LIN {X 0,Y 418.536,Z 472.34,A -85,B 0,C 180,E1 -10078.075,E2 -10078.075} C_VEL
LIN {X 0,Y 418.665,Z 472.33,A -85,B 0,C 180,E1 -10080,E2 -10080} C_VEL
LIN {X 0,Y 418.503,Z 472.347,A -85,B 0,C 180,E1 -10082.888,E2 -10082.888} C_VEL
LIN {X 0,Y 418.524,Z 472.35,A -85,B 0,C 180,E1 -10085.783,E2 -10085.783} C_VEL
LIN {X 0,Y 418.391,Z 472.364,A -85,B 0,C 180,E1 -10088.695,E2 -10088.695} C_VEL
LIN {X 0,Y 418.307,Z 472.371,A -85,B 0,C 180,E1 -10091.631,E2 -10091.631} C_VEL
LIN {X 0,Y 418.293,Z 472.377,A -85,B 0,C 180,E1 -10094.597,E2 -10094.597} C_VEL
LIN {X 0,Y 418.279,Z 472.366,A -85,B 0,C 180,E1 -10097.604,E2 -10097.604} C_VEL
LIN {X 0,Y 418.242,Z 472.376,A -85,B 0,C 180,E1 -10100.663,E2 -10100.663} C_VEL
LIN {X 0,Y 418.28,Z 472.382,A -85,B 0,C 180,E1 -10103.782,E2 -10103.782} C_VEL
LIN {X 0,Y 418.303,Z 472.362,A -85,B 0,C 180,E1 -10107.071,E2 -10107.071} C_VEL
LIN {X 0,Y 418.256,Z 472.383,A -85,B 0,C 180,E1 -10110.271,E2 -10110.271} C_VEL
LIN {X 0,Y 418.243,Z 472.378,A -85,B 0,C 180,E1 -10113.678,E2 -10113.678} C_VEL
LIN {X 0,Y 418.24,Z 472.385,A -85,B 0,C 180,E1 -10117.224,E2 -10117.224} C_VEL
LIN {X 0,Y 418.25,Z 472.386,A -85,B 0,C 180,E1 -10119.682,E2 -10119.682} C_VEL
LIN {X 0,Y 418.225,Z 472.377,A -85,B 0,C 180,E1 -10122.322,E2 -10122.322} C_VEL
LIN {X 0,Y 418.254,Z 472.371,A -85,B 0,C 180,E1 -10125.113,E2 -10125.113} C_VEL
LIN {X 0,Y 418.289,Z 472.38,A -85,B 0,C 180,E1 -10127.774,E2 -10127.774} C_VEL
LIN {X 0,Y 418.262,Z 472.385,A -85,B 0,C 180,E1 -10131.56,E2 -10131.56} C_VEL
LIN {X 0,Y 418.258,Z 472.386,A -85,B 0,C 180,E1 -10135.16,E2 -10135.16} C_VEL
LIN {X 0,Y 418.282,Z 472.582,A -85,B 0,C 180,E1 -10137.69,E2 -10137.69} C_VEL
LIN {X 0,Y 421.773,Z 487.467,A -85,B 0,C 180,E1 -10140.305,E2 -10140.305} C_VEL
LIN {X 0,Y 423.139,Z 494.876,A -85,B 0,C 180,E1 -10141.54,E2 -10141.54} C_VEL
LIN {X 0,Y 421.976,Z 513.448,A -85,B 0,C 180,E1 -10144.341,E2 -10144.341} C_VEL
LIN {X 0,Y 420.64,Z 535.68,A -85,B 0,C 180,E1 -10147.66,E2 -10147.66} C_VEL
LIN {X 0,Y 419.505,Z 557.237,A -85,B 0,C 180,E1 -10150.87,E2 -10150.87} C_VEL
LIN {X 0,Y 422.696,Z 586.903,A -85,B 0,C 180,E1 -10151.56,E2 -10151.56} C_VEL
LIN {X 0,Y 423.368,Z 594.694,A -85,B 0,C 180,E1 -10151.724,E2 -10151.724} C_VEL
LIN {X 0,Y 422.593,Z 667.918,A -85,B 0,C 180,E1 -10152.987,E2 -10152.987} C_VEL
LIN {X 0,Y 422.008,Z 681.219,A -85,B 0,C 180,E1 -10153.399,E2 -10153.399} C_VEL
LIN {X 0,Y 421.231,Z 694.57,A -85,B 0,C 180,E1 -10154.021,E2 -10154.021} C_VEL
LIN {X 0,Y 420.554,Z 705.824,A -85,B 0,C 180,E1 -10154.74,E2 -10154.74} C_VEL
LIN {X 0,Y 419.697,Z 717.543,A -85,B 0,C 180,E1 -10155.701,E2 -10155.701} C_VEL
LIN {X 0,Y 419.002,Z 727.885,A -85,B 0,C 180,E1 -10156.761,E2 -10156.761} C_VEL
LIN {X 0,Y 418.593,Z 735.017,A -85,B 0,C 180,E1 -10157.64,E2 -10157.64} C_VEL
LIN {X 0,Y 418.002,Z 744.878,A -85,B 0,C 180,E1 -10159.097,E2 -10159.097} C_VEL
LIN {X 0,Y 417.68,Z 752.774,A -85,B 0,C 180,E1 -10160.558,E2 -10160.558} C_VEL
LIN {X 0,Y 417.506,Z 760.077,A -85,B 0,C 180,E1 -10162.261,E2 -10162.261} C_VEL
LIN {X 0,Y 417.494,Z 764.689,A -85,B 0,C 180,E1 -10163.63,E2 -10163.63} C_VEL
LIN {X 0,Y 417.619,Z 768.711,A -85,B 0,C 180,E1 -10165.173,E2 -10165.173} C_VEL
LIN {X 0,Y 417.674,Z 770.646,A -85,B 0,C 180,E1 -10166.141,E2 -10166.141} C_VEL
LIN {X 0,Y 417.648,Z 772.089,A -85,B 0,C 180,E1 -10167.106,E2 -10167.106} C_VEL
LIN {X 0,Y 417.907,Z 773.786,A -85,B 0,C 180,E1 -10169.036,E2 -10169.036} C_VEL
LIN {X 0,Y 417.924,Z 774.012,A -85,B 0,C 180,E1 -10170,E2 -10170} C_VEL
LIN {X 0,Y 417.907,Z 773.785,A -85,B 0,C 180,E1 -10170.964,E2 -10170.964} C_VEL
LIN {X 0,Y 417.648,Z 772.089,A -85,B 0,C 180,E1 -10172.894,E2 -10172.894} C_VEL
LIN {X 0,Y 417.674,Z 770.645,A -85,B 0,C 180,E1 -10173.859,E2 -10173.859} C_VEL
LIN {X 0,Y 417.534,Z 767.586,A -85,B 0,C 180,E1 -10175.312,E2 -10175.312} C_VEL
LIN {X 0,Y 417.475,Z 763.466,A -85,B 0,C 180,E1 -10176.767,E2 -10176.767} C_VEL
LIN {X 0,Y 417.531,Z 757.153,A -85,B 0,C 180,E1 -10178.469,E2 -10178.469} C_VEL
LIN {X 0,Y 417.723,Z 750.287,A -85,B 0,C 180,E1 -10179.93,E2 -10179.93} C_VEL
LIN {X 0,Y 418.17,Z 741.814,A -85,B 0,C 180,E1 -10181.389,E2 -10181.389} C_VEL
LIN {X 0,Y 418.764,Z 733.161,A -85,B 0,C 180,E1 -10182.602,E2 -10182.602} C_VEL
LIN {X 0,Y 419.355,Z 722.483,A -85,B 0,C 180,E1 -10183.816,E2 -10183.816} C_VEL
LIN {X 0,Y 420.141,Z 710.52,A -85,B 0,C 180,E1 -10184.903,E2 -10184.903} C_VEL
LIN {X 0,Y 421.03,Z 698.539,A -85,B 0,C 180,E1 -10185.738,E2 -10185.738} C_VEL
LIN {X 0,Y 421.752,Z 686.096,A -85,B 0,C 180,E1 -10186.394,E2 -10186.394} C_VEL
LIN {X 0,Y 422.39,Z 673.352,A -85,B 0,C 180,E1 -10186.866,E2 -10186.866} C_VEL
LIN {X 0,Y 422.723,Z 658.22,A -85,B 0,C 180,E1 -10187.194,E2 -10187.194} C_VEL
LIN {X 0,Y 423.312,Z 592.38,A -85,B 0,C 180,E1 -10188.314,E2 -10188.314} C_VEL
LIN {X 0,Y 419.505,Z 557.278,A -85,B 0,C 180,E1 -10189.121,E2 -10189.121} C_VEL
LIN {X 0,Y 420.722,Z 533.922,A -85,B 0,C 180,E1 -10192.594,E2 -10192.594} C_VEL
LIN {X 0,Y 422.251,Z 509.398,A -85,B 0,C 180,E1 -10196.258,E2 -10196.258} C_VEL
LIN {X 0,Y 423.139,Z 494.649,A -85,B 0,C 180,E1 -10198.486,E2 -10198.486} C_VEL
LIN {X 0,Y 421.349,Z 485.456,A -85,B 0,C 180,E1 -10200.025,E2 -10200.025} C_VEL
LIN {X 0,Y 418.28,Z 472.498,A -85,B 0,C 180,E1 -10202.346,E2 -10202.346} C_VEL
LIN {X 0,Y 418.257,Z 472.387,A -85,B 0,C 180,E1 -10204.84,E2 -10204.84} C_VEL
LIN {X 0,Y 418.262,Z 472.385,A -85,B 0,C 180,E1 -10208.44,E2 -10208.44} C_VEL
LIN {X 0,Y 418.289,Z 472.381,A -85,B 0,C 180,E1 -10212.226,E2 -10212.226} C_VEL
LIN {X 0,Y 418.247,Z 472.37,A -85,B 0,C 180,E1 -10215.11,E2 -10215.11} C_VEL
LIN {X 0,Y 418.235,Z 472.376,A -85,B 0,C 180,E1 -10217.766,E2 -10217.766} C_VEL
LIN {X 0,Y 418.254,Z 472.381,A -85,B 0,C 180,E1 -10220.617,E2 -10220.617} C_VEL
LIN {X 0,Y 418.24,Z 472.387,A -85,B 0,C 180,E1 -10223.975,E2 -10223.975} C_VEL
LIN {X 0,Y 418.251,Z 472.375,A -85,B 0,C 180,E1 -10227.155,E2 -10227.155} C_VEL
LIN {X 0,Y 418.268,Z 472.379,A -85,B 0,C 180,E1 -10230.838,E2 -10230.838} C_VEL
LIN {X 0,Y 418.264,Z 472.371,A -85,B 0,C 180,E1 -10234.095,E2 -10234.095} C_VEL
LIN {X 0,Y 418.23,Z 472.385,A -85,B 0,C 180,E1 -10237.263,E2 -10237.263} C_VEL
LIN {X 0,Y 418.275,Z 472.364,A -85,B 0,C 180,E1 -10240.364,E2 -10240.364} C_VEL
LIN {X 0,Y 418.308,Z 472.37,A -85,B 0,C 180,E1 -10243.404,E2 -10243.404} C_VEL
LIN {X 0,Y 418.337,Z 472.37,A -85,B 0,C 180,E1 -10246.999,E2 -10246.999} C_VEL
LIN {X 0,Y 418.333,Z 472.369,A -85,B 0,C 180,E1 -10250.328,E2 -10250.328} C_VEL
LIN {X 0,Y 418.486,Z 472.352,A -85,B 0,C 180,E1 -10253.249,E2 -10253.249} C_VEL
LIN {X 0,Y 418.337,Z 472.361,A -85,B 0,C 180,E1 -10255.182,E2 -10255.182} C_VEL
LIN {X 0,Y 418.536,Z 472.346,A -85,B 0,C 180,E1 -10258.075,E2 -10258.075} C_VEL
LIN {X 0,Y 418.665,Z 472.332,A -85,B 0,C 180,E1 -10260,E2 -10260} C_VEL
LIN {X 0,Y 418.503,Z 472.345,A -85,B 0,C 180,E1 -10262.888,E2 -10262.888} C_VEL
LIN {X 0,Y 418.484,Z 472.355,A -85,B 0,C 180,E1 -10266.615,E2 -10266.615} C_VEL
LIN {X 0,Y 418.333,Z 472.361,A -85,B 0,C 180,E1 -10269.672,E2 -10269.672} C_VEL
LIN {X 0,Y 418.338,Z 472.374,A -85,B 0,C 180,E1 -10273.001,E2 -10273.001} C_VEL
LIN {X 0,Y 418.304,Z 472.371,A -85,B 0,C 180,E1 -10276.736,E2 -10276.736} C_VEL
LIN {X 0,Y 418.263,Z 472.381,A -85,B 0,C 180,E1 -10279.791,E2 -10279.791} C_VEL
LIN {X 0,Y 418.23,Z 472.381,A -85,B 0,C 180,E1 -10282.737,E2 -10282.737} C_VEL
LIN {X 0,Y 418.264,Z 472.381,A -85,B 0,C 180,E1 -10285.905,E2 -10285.905} C_VEL
LIN {X 0,Y 418.268,Z 472.36,A -85,B 0,C 180,E1 -10289.162,E2 -10289.162} C_VEL
LIN {X 0,Y 418.252,Z 472.37,A -85,B 0,C 180,E1 -10292.845,E2 -10292.845} C_VEL
LIN {X 0,Y 418.243,Z 472.385,A -85,B 0,C 180,E1 -10296.239,E2 -10296.239} C_VEL
LIN {X 0,Y 418.24,Z 472.361,A -85,B 0,C 180,E1 -10299.683,E2 -10299.683} C_VEL
LIN {X 0,Y 418.225,Z 472.38,A -85,B 0,C 180,E1 -10302.322,E2 -10302.322} C_VEL
LIN {X 0,Y 418.235,Z 472.385,A -85,B 0,C 180,E1 -10305.11,E2 -10305.11} C_VEL
LIN {X 0,Y 418.239,Z 472.372,A -85,B 0,C 180,E1 -10307.768,E2 -10307.768} C_VEL
LIN {X 0,Y 418.259,Z 472.385,A -85,B 0,C 180,E1 -10310.619,E2 -10310.619} C_VEL
LIN {X 0,Y 418.244,Z 472.359,A -85,B 0,C 180,E1 -10313.977,E2 -10313.977} C_VEL
LIN {X 0,Y 418.257,Z 472.359,A -85,B 0,C 180,E1 -10317.157,E2 -10317.157} C_VEL
LIN {X 0,Y 418.268,Z 472.378,A -85,B 0,C 180,E1 -10320.896,E2 -10320.896} C_VEL
LIN {X 0,Y 418.271,Z 472.368,A -85,B 0,C 180,E1 -10324.097,E2 -10324.097} C_VEL
LIN {X 0,Y 418.239,Z 472.371,A -85,B 0,C 180,E1 -10327.265,E2 -10327.265} C_VEL
LIN {X 0,Y 418.324,Z 472.346,A -85,B 0,C 180,E1 -10330.877,E2 -10330.877} C_VEL
LIN {X 0,Y 418.375,Z 472.623,A -85,B 0,C 180,E1 -10331.261,E2 -10331.261} C_VEL
LIN {X 0,Y 418.655,Z 473.76,A -85,B 0,C 180,E1 -10331.401,E2 -10331.401} C_VEL
LIN {X 0,Y 424.299,Z 488.537,A -85,B 0,C 180,E1 -10331.94,E2 -10331.94} C_VEL
LIN {X 0,Y 423.71,Z 551.851,A -85,B 0,C 180,E1 -10333.033,E2 -10333.033} C_VEL
LIN {X 0,Y 423.641,Z 564.47,A -85,B 0,C 180,E1 -10333.403,E2 -10333.403} C_VEL
LIN {X 0,Y 423.281,Z 577.262,A -85,B 0,C 180,E1 -10333.977,E2 -10333.977} C_VEL
LIN {X 0,Y 422.895,Z 589.004,A -85,B 0,C 180,E1 -10334.702,E2 -10334.702} C_VEL
LIN {X 0,Y 422.287,Z 599.691,A -85,B 0,C 180,E1 -10335.544,E2 -10335.544} C_VEL
LIN {X 0,Y 421.612,Z 610.545,A -85,B 0,C 180,E1 -10336.627,E2 -10336.627} C_VEL
LIN {X 0,Y 420.921,Z 621.071,A -85,B 0,C 180,E1 -10337.954,E2 -10337.954} C_VEL
LIN {X 0,Y 420.413,Z 628.814,A -85,B 0,C 180,E1 -10339.16,E2 -10339.16} C_VEL
LIN {X 0,Y 419.767,Z 636.5,A -85,B 0,C 180,E1 -10340.63,E2 -10340.63} C_VEL
LIN {X 0,Y 419.323,Z 642.255,A -85,B 0,C 180,E1 -10342.003,E2 -10342.003} C_VEL
LIN {X 0,Y 419.063,Z 646.526,A -85,B 0,C 180,E1 -10343.258,E2 -10343.258} C_VEL
LIN {X 0,Y 418.621,Z 650.42,A -85,B 0,C 180,E1 -10344.702,E2 -10344.702} C_VEL
LIN {X 0,Y 418.398,Z 652.498,A -85,B 0,C 180,E1 -10345.73,E2 -10345.73} C_VEL
LIN {X 0,Y 417.639,Z 653.952,A -85,B 0,C 180,E1 -10346.509,E2 -10346.509} C_VEL
LIN {X 0,Y 414.72,Z 655.903,A -85,B 0,C 180,E1 -10347.785,E2 -10347.785} C_VEL
LIN {X 0,Y 412.318,Z 656.955,A -85,B 0,C 180,E1 -10348.826,E2 -10348.826} C_VEL
LIN {X 0,Y 411.309,Z 657.36,A -85,B 0,C 180,E1 -10349.635,E2 -10349.635} C_VEL
LIN {X 0,Y 411.236,Z 657.406,A -85,B 0,C 180,E1 -10349.91,E2 -10349.91} C_VEL
LIN {X 0,Y 411.256,Z 657.243,A -85,B 0,C 180,E1 -10350.979,E2 -10350.979} C_VEL
LIN {X 0,Y 411.181,Z 656.69,A -85,B 0,C 180,E1 -10351.959,E2 -10351.959} C_VEL
LIN {X 0,Y 411.339,Z 655.735,A -85,B 0,C 180,E1 -10352.938,E2 -10352.938} C_VEL
LIN {X 0,Y 411.318,Z 654.429,A -85,B 0,C 180,E1 -10353.919,E2 -10353.919} C_VEL
LIN {X 0,Y 411.614,Z 651.618,A -85,B 0,C 180,E1 -10355.388,E2 -10355.388} C_VEL
LIN {X 0,Y 412.065,Z 647.796,A -85,B 0,C 180,E1 -10356.857,E2 -10356.857} C_VEL
LIN {X 0,Y 412.366,Z 642.722,A -85,B 0,C 180,E1 -10358.378,E2 -10358.378} C_VEL
LIN {X 0,Y 412.913,Z 636.698,A -85,B 0,C 180,E1 -10359.8,E2 -10359.8} C_VEL
LIN {X 0,Y 413.612,Z 628.922,A -85,B 0,C 180,E1 -10361.268,E2 -10361.268} C_VEL
LIN {X 0,Y 414.28,Z 619.255,A -85,B 0,C 180,E1 -10362.74,E2 -10362.74} C_VEL
LIN {X 0,Y 414.951,Z 610.219,A -85,B 0,C 180,E1 -10363.841,E2 -10363.841} C_VEL
LIN {X 0,Y 415.667,Z 599.725,A -85,B 0,C 180,E1 -10364.873,E2 -10364.873} C_VEL
LIN {X 0,Y 416.209,Z 588.069,A -85,B 0,C 180,E1 -10365.787,E2 -10365.787} C_VEL
LIN {X 0,Y 416.646,Z 576.642,A -85,B 0,C 180,E1 -10366.474,E2 -10366.474} C_VEL
LIN {X 0,Y 416.932,Z 563.782,A -85,B 0,C 180,E1 -10367.03,E2 -10367.03} C_VEL
LIN {X 0,Y 416.972,Z 551.522,A -85,B 0,C 180,E1 -10367.376,E2 -10367.376} C_VEL
LIN {X 0,Y 417.43,Z 489.383,A -85,B 0,C 180,E1 -10368.47,E2 -10368.47} C_VEL
LIN {X 0,Y 411.516,Z 474.325,A -85,B 0,C 180,E1 -10369.052,E2 -10369.052} C_VEL
LIN {X 0,Y 411.297,Z 473.373,A -85,B 0,C 180,E1 -10369.236,E2 -10369.236} C_VEL
LIN {X 0,Y 411.204,Z 473.25,A -85,B 0,C 180,E1 -10373.147,E2 -10373.147} C_VEL
LIN {X 0,Y 411.238,Z 473.237,A -85,B 0,C 180,E1 -10376.38,E2 -10376.38} C_VEL
LIN {X 0,Y 411.2,Z 473.263,A -85,B 0,C 180,E1 -10379.712,E2 -10379.712} C_VEL
LIN {X 0,Y 411.205,Z 473.259,A -85,B 0,C 180,E1 -10383.155,E2 -10383.155} C_VEL
LIN {X 0,Y 411.194,Z 473.256,A -85,B 0,C 180,E1 -10386.552,E2 -10386.552} C_VEL
LIN {X 0,Y 411.214,Z 473.262,A -85,B 0,C 180,E1 -10389.727,E2 -10389.727} C_VEL
LIN {X 0,Y 411.174,Z 473.253,A -85,B 0,C 180,E1 -10393.132,E2 -10393.132} C_VEL
LIN {X 0,Y 411.165,Z 473.267,A -85,B 0,C 180,E1 -10395.88,E2 -10395.88} C_VEL
LIN {X 0,Y 411.159,Z 473.254,A -85,B 0,C 180,E1 -10398.771,E2 -10398.771} C_VEL
LIN {X 0,Y 411.191,Z 473.256,A -85,B 0,C 180,E1 -10402.026,E2 -10402.026} C_VEL
LIN {X 0,Y 411.2,Z 473.258,A -85,B 0,C 180,E1 -10405.666,E2 -10405.666} C_VEL
LIN {X 0,Y 411.191,Z 473.233,A -85,B 0,C 180,E1 -10409.152,E2 -10409.152} C_VEL
LIN {X 0,Y 411.253,Z 473.247,A -85,B 0,C 180,E1 -10412.522,E2 -10412.522} C_VEL
LIN {X 0,Y 411.219,Z 473.257,A -85,B 0,C 180,E1 -10415.784,E2 -10415.784} C_VEL
LIN {X 0,Y 411.188,Z 473.259,A -85,B 0,C 180,E1 -10418.965,E2 -10418.965} C_VEL
LIN {X 0,Y 411.244,Z 473.252,A -85,B 0,C 180,E1 -10422.084,E2 -10422.084} C_VEL
LIN {X 0,Y 411.252,Z 473.251,A -85,B 0,C 180,E1 -10425.147,E2 -10425.147} C_VEL
LIN {X 0,Y 411.276,Z 473.25,A -85,B 0,C 180,E1 -10428.167,E2 -10428.167} C_VEL
LIN {X 0,Y 411.473,Z 473.223,A -85,B 0,C 180,E1 -10432.146,E2 -10432.146} C_VEL
LIN {X 0,Y 411.466,Z 473.226,A -85,B 0,C 180,E1 -10434.118,E2 -10434.118} C_VEL
LIN {X 0,Y 411.505,Z 473.216,A -85,B 0,C 180,E1 -10438.042,E2 -10438.042} C_VEL
LIN {X 0,Y 411.635,Z 473.206,A -85,B 0,C 180,E1 -10440,E2 -10440} C_VEL
LIN {X 0,Y 411.458,Z 473.225,A -85,B 0,C 180,E1 -10442.937,E2 -10442.937} C_VEL
LIN {X 0,Y 411.483,Z 473.226,A -85,B 0,C 180,E1 -10445.882,E2 -10445.882} C_VEL
LIN {X 0,Y 411.346,Z 473.242,A -85,B 0,C 180,E1 -10448.845,E2 -10448.845} C_VEL
LIN {X 0,Y 411.276,Z 473.249,A -85,B 0,C 180,E1 -10451.833,E2 -10451.833} C_VEL
LIN {X 0,Y 411.251,Z 473.255,A -85,B 0,C 180,E1 -10454.853,E2 -10454.853} C_VEL
LIN {X 0,Y 411.244,Z 473.238,A -85,B 0,C 180,E1 -10457.915,E2 -10457.915} C_VEL
LIN {X 0,Y 411.188,Z 473.256,A -85,B 0,C 180,E1 -10461.035,E2 -10461.035} C_VEL
LIN {X 0,Y 411.219,Z 473.257,A -85,B 0,C 180,E1 -10464.216,E2 -10464.216} C_VEL
LIN {X 0,Y 411.253,Z 473.242,A -85,B 0,C 180,E1 -10467.478,E2 -10467.478} C_VEL
LIN {X 0,Y 411.194,Z 473.262,A -85,B 0,C 180,E1 -10470.847,E2 -10470.847} C_VEL
LIN {X 0,Y 411.201,Z 473.26,A -85,B 0,C 180,E1 -10474.334,E2 -10474.334} C_VEL
LIN {X 0,Y 411.195,Z 473.258,A -85,B 0,C 180,E1 -10477.974,E2 -10477.974} C_VEL
LIN {X 0,Y 411.178,Z 473.265,A -85,B 0,C 180,E1 -10480.505,E2 -10480.505} C_VEL
LIN {X 0,Y 411.168,Z 473.25,A -85,B 0,C 180,E1 -10483.134,E2 -10483.134} C_VEL
LIN {X 0,Y 411.232,Z 473.253,A -85,B 0,C 180,E1 -10485.872,E2 -10485.872} C_VEL
LIN {X 0,Y 411.207,Z 473.254,A -85,B 0,C 180,E1 -10488.765,E2 -10488.765} C_VEL
LIN {X 0,Y 411.201,Z 473.264,A -85,B 0,C 180,E1 -10492.028,E2 -10492.028} C_VEL
LIN {X 0,Y 411.204,Z 473.261,A -85,B 0,C 180,E1 -10495.667,E2 -10495.667} C_VEL
LIN {X 0,Y 411.241,Z 473.427,A -85,B 0,C 180,E1 -10497.358,E2 -10497.358} C_VEL
LIN {X 0,Y 414.904,Z 489.081,A -85,B 0,C 180,E1 -10500.172,E2 -10500.172} C_VEL
LIN {X 0,Y 416.266,Z 496.273,A -85,B 0,C 180,E1 -10501.395,E2 -10501.395} C_VEL
LIN {X 0,Y 415.073,Z 514.231,A -85,B 0,C 180,E1 -10504.152,E2 -10504.152} C_VEL
LIN {X 0,Y 413.65,Z 536.399,A -85,B 0,C 180,E1 -10507.526,E2 -10507.526} C_VEL
LIN {X 0,Y 412.575,Z 556.343,A -85,B 0,C 180,E1 -10510.545,E2 -10510.545} C_VEL
LIN {X 0,Y 415.931,Z 587.374,A -85,B 0,C 180,E1 -10511.274,E2 -10511.274} C_VEL
LIN {X 0,Y 416.594,Z 595.875,A -85,B 0,C 180,E1 -10511.454,E2 -10511.454} C_VEL
LIN {X 0,Y 415.799,Z 666.93,A -85,B 0,C 180,E1 -10512.7,E2 -10512.7} C_VEL
LIN {X 0,Y 415.202,Z 680.228,A -85,B 0,C 180,E1 -10513.119,E2 -10513.119} C_VEL
LIN {X 0,Y 414.376,Z 693.573,A -85,B 0,C 180,E1 -10513.749,E2 -10513.749} C_VEL
LIN {X 0,Y 413.631,Z 704.819,A -85,B 0,C 180,E1 -10514.478,E2 -10514.478} C_VEL
LIN {X 0,Y 412.746,Z 716.537,A -85,B 0,C 180,E1 -10515.455,E2 -10515.455} C_VEL
LIN {X 0,Y 412.018,Z 726.405,A -85,B 0,C 180,E1 -10516.478,E2 -10516.478} C_VEL
LIN {X 0,Y 411.638,Z 734.018,A -85,B 0,C 180,E1 -10517.427,E2 -10517.427} C_VEL
LIN {X 0,Y 411.052,Z 742.351,A -85,B 0,C 180,E1 -10518.661,E2 -10518.661} C_VEL
LIN {X 0,Y 410.637,Z 750.568,A -85,B 0,C 180,E1 -10520.146,E2 -10520.146} C_VEL
LIN {X 0,Y 410.451,Z 757.194,A -85,B 0,C 180,E1 -10521.632,E2 -10521.632} C_VEL
LIN {X 0,Y 410.418,Z 763.067,A -85,B 0,C 180,E1 -10523.312,E2 -10523.312} C_VEL
LIN {X 0,Y 410.546,Z 767.714,A -85,B 0,C 180,E1 -10525.09,E2 -10525.09} C_VEL
LIN {X 0,Y 410.635,Z 769.655,A -85,B 0,C 180,E1 -10526.075,E2 -10526.075} C_VEL
LIN {X 0,Y 410.604,Z 771.098,A -85,B 0,C 180,E1 -10527.057,E2 -10527.057} C_VEL
LIN {X 0,Y 410.88,Z 772.798,A -85,B 0,C 180,E1 -10529.02,E2 -10529.02} C_VEL
LIN {X 0,Y 410.902,Z 773.025,A -85,B 0,C 180,E1 -10530,E2 -10530} C_VEL
LIN {X 0,Y 410.881,Z 772.797,A -85,B 0,C 180,E1 -10530.98,E2 -10530.98} C_VEL
LIN {X 0,Y 410.604,Z 771.097,A -85,B 0,C 180,E1 -10532.943,E2 -10532.943} C_VEL
LIN {X 0,Y 410.635,Z 769.653,A -85,B 0,C 180,E1 -10533.925,E2 -10533.925} C_VEL
LIN {X 0,Y 410.46,Z 766.587,A -85,B 0,C 180,E1 -10535.404,E2 -10535.404} C_VEL
LIN {X 0,Y 410.421,Z 762.466,A -85,B 0,C 180,E1 -10536.884,E2 -10536.884} C_VEL
LIN {X 0,Y 410.464,Z 756.147,A -85,B 0,C 180,E1 -10538.616,E2 -10538.616} C_VEL
LIN {X 0,Y 410.665,Z 749.278,A -85,B 0,C 180,E1 -10540.103,E2 -10540.103} C_VEL
LIN {X 0,Y 411.145,Z 740.804,A -85,B 0,C 180,E1 -10541.586,E2 -10541.586} C_VEL
LIN {X 0,Y 411.774,Z 732.151,A -85,B 0,C 180,E1 -10542.819,E2 -10542.819} C_VEL
LIN {X 0,Y 412.319,Z 722.665,A -85,B 0,C 180,E1 -10543.931,E2 -10543.931} C_VEL
LIN {X 0,Y 413.112,Z 710.953,A -85,B 0,C 180,E1 -10545.036,E2 -10545.036} C_VEL
LIN {X 0,Y 414.041,Z 699.479,A -85,B 0,C 180,E1 -10545.885,E2 -10545.885} C_VEL
LIN {X 0,Y 414.765,Z 687.701,A -85,B 0,C 180,E1 -10546.551,E2 -10546.551} C_VEL
LIN {X 0,Y 415.503,Z 674.18,A -85,B 0,C 180,E1 -10547.09,E2 -10547.09} C_VEL
LIN {X 0,Y 415.893,Z 660.789,A -85,B 0,C 180,E1 -10547.422,E2 -10547.422} C_VEL
LIN {X 0,Y 416.518,Z 592.858,A -85,B 0,C 180,E1 -10548.597,E2 -10548.597} C_VEL
LIN {X 0,Y 412.55,Z 556.589,A -85,B 0,C 180,E1 -10549.433,E2 -10549.433} C_VEL
LIN {X 0,Y 412.898,Z 549.484,A -85,B 0,C 180,E1 -10550.47,E2 -10550.47} C_VEL
LIN {X 0,Y 414.285,Z 526.14,A -85,B 0,C 180,E1 -10554.025,E2 -10554.025} C_VEL
LIN {X 0,Y 415.776,Z 503.859,A -85,B 0,C 180,E1 -10557.426,E2 -10557.426} C_VEL
LIN {X 0,Y 416.271,Z 496.209,A -85,B 0,C 180,E1 -10558.606,E2 -10558.606} C_VEL
LIN {X 0,Y 414.493,Z 487.187,A -85,B 0,C 180,E1 -10560.147,E2 -10560.147} C_VEL
LIN {X 0,Y 411.226,Z 473.379,A -85,B 0,C 180,E1 -10562.661,E2 -10562.661} C_VEL
LIN {X 0,Y 411.197,Z 473.26,A -85,B 0,C 180,E1 -10565.528,E2 -10565.528} C_VEL
LIN {X 0,Y 411.227,Z 473.255,A -85,B 0,C 180,E1 -10569.222,E2 -10569.222} C_VEL
LIN {X 0,Y 411.229,Z 473.262,A -85,B 0,C 180,E1 -10572.703,E2 -10572.703} C_VEL
LIN {X 0,Y 411.167,Z 473.244,A -85,B 0,C 180,E1 -10575.88,E2 -10575.88} C_VEL
LIN {X 0,Y 411.16,Z 473.269,A -85,B 0,C 180,E1 -10578.771,E2 -10578.771} C_VEL
LIN {X 0,Y 411.206,Z 473.255,A -85,B 0,C 180,E1 -10581.83,E2 -10581.83} C_VEL
LIN {X 0,Y 411.205,Z 473.258,A -85,B 0,C 180,E1 -10585.121,E2 -10585.121} C_VEL
LIN {X 0,Y 411.162,Z 473.261,A -85,B 0,C 180,E1 -10588.002,E2 -10588.002} C_VEL
LIN {X 0,Y 411.217,Z 473.255,A -85,B 0,C 180,E1 -10591.41,E2 -10591.41} C_VEL
LIN {X 0,Y 411.231,Z 473.243,A -85,B 0,C 180,E1 -10593.619,E2 -10593.619} C_VEL
LIN {X 0,Y 411.195,Z 473.263,A -85,B 0,C 180,E1 -10596.852,E2 -10596.852} C_VEL
LIN {X 0,Y 411.207,Z 473.248,A -85,B 0,C 180,E1 -10600.05,E2 -10600.05} C_VEL
LIN {X 0,Y 411.255,Z 473.25,A -85,B 0,C 180,E1 -10603.131,E2 -10603.131} C_VEL
LIN {X 0,Y 411.297,Z 473.248,A -85,B 0,C 180,E1 -10606.896,E2 -10606.896} C_VEL
LIN {X 0,Y 411.285,Z 473.245,A -85,B 0,C 180,E1 -10610.161,E2 -10610.161} C_VEL
LIN {X 0,Y 411.449,Z 473.229,A -85,B 0,C 180,E1 -10613.133,E2 -10613.133} C_VEL
LIN {X 0,Y 411.308,Z 473.237,A -85,B 0,C 180,E1 -10615.099,E2 -10615.099} C_VEL
LIN {X 0,Y 411.505,Z 473.222,A -85,B 0,C 180,E1 -10618.043,E2 -10618.043} C_VEL
LIN {X 0,Y 411.635,Z 473.208,A -85,B 0,C 180,E1 -10620,E2 -10620} C_VEL
LIN {X 0,Y 411.459,Z 473.222,A -85,B 0,C 180,E1 -10622.937,E2 -10622.937} C_VEL
LIN {X 0,Y 411.447,Z 473.229,A -85,B 0,C 180,E1 -10626.614,E2 -10626.614} C_VEL
LIN {X 0,Y 411.285,Z 473.239,A -85,B 0,C 180,E1 -10629.839,E2 -10629.839} C_VEL
LIN {X 0,Y 411.297,Z 473.25,A -85,B 0,C 180,E1 -10633.104,E2 -10633.104} C_VEL
LIN {X 0,Y 411.249,Z 473.251,A -85,B 0,C 180,E1 -10636.889,E2 -10636.889} C_VEL
LIN {X 0,Y 411.223,Z 473.258,A -85,B 0,C 180,E1 -10639.987,E2 -10639.987} C_VEL
LIN {X 0,Y 411.196,Z 473.261,A -85,B 0,C 180,E1 -10643.148,E2 -10643.148} C_VEL
LIN {X 0,Y 411.231,Z 473.259,A -85,B 0,C 180,E1 -10646.382,E2 -10646.382} C_VEL
LIN {X 0,Y 411.204,Z 473.236,A -85,B 0,C 180,E1 -10649.713,E2 -10649.713} C_VEL
LIN {X 0,Y 411.201,Z 473.253,A -85,B 0,C 180,E1 -10653.157,E2 -10653.157} C_VEL
LIN {X 0,Y 411.19,Z 473.266,A -85,B 0,C 180,E1 -10656.554,E2 -10656.554} C_VEL
LIN {X 0,Y 411.204,Z 473.236,A -85,B 0,C 180,E1 -10659.728,E2 -10659.728} C_VEL
LIN {X 0,Y 411.169,Z 473.269,A -85,B 0,C 180,E1 -10663.134,E2 -10663.134} C_VEL
LIN {X 0,Y 411.169,Z 473.259,A -85,B 0,C 180,E1 -10665.881,E2 -10665.881} C_VEL
LIN {X 0,Y 411.163,Z 473.259,A -85,B 0,C 180,E1 -10668.772,E2 -10668.772} C_VEL
LIN {X 0,Y 411.21,Z 473.256,A -85,B 0,C 180,E1 -10671.831,E2 -10671.831} C_VEL
LIN {X 0,Y 411.21,Z 473.217,A -85,B 0,C 180,E1 -10675.122,E2 -10675.122} C_VEL
LIN {X 0,Y 411.165,Z 473.261,A -85,B 0,C 180,E1 -10678.004,E2 -10678.004} C_VEL
LIN {X 0,Y 411.218,Z 473.248,A -85,B 0,C 180,E1 -10681.411,E2 -10681.411} C_VEL
LIN {X 0,Y 411.238,Z 473.236,A -85,B 0,C 180,E1 -10683.62,E2 -10683.62} C_VEL
LIN {X 0,Y 411.204,Z 473.251,A -85,B 0,C 180,E1 -10686.853,E2 -10686.853} C_VEL
LIN {X 0,Y 411.308,Z 473.339,A -85,B 0,C 180,E1 -10690.862,E2 -10690.862} C_VEL
LIN {X 0,Y 411.456,Z 474.138,A -85,B 0,C 180,E1 -10691.031,E2 -10691.031} C_VEL
LIN {X 0,Y 417.419,Z 489.367,A -85,B 0,C 180,E1 -10691.628,E2 -10691.628} C_VEL
LIN {X 0,Y 416.975,Z 554.337,A -85,B 0,C 180,E1 -10692.782,E2 -10692.782} C_VEL
LIN {X 0,Y 416.801,Z 567.775,A -85,B 0,C 180,E1 -10693.217,E2 -10693.217} C_VEL
LIN {X 0,Y 416.499,Z 580.488,A -85,B 0,C 180,E1 -10693.835,E2 -10693.835} C_VEL
LIN {X 0,Y 416.078,Z 591.709,A -85,B 0,C 180,E1 -10694.57,E2 -10694.57} C_VEL
LIN {X 0,Y 415.34,Z 603.297,A -85,B 0,C 180,E1 -10695.547,E2 -10695.547} C_VEL
LIN {X 0,Y 414.661,Z 613.632,A -85,B 0,C 180,E1 -10696.649,E2 -10696.649} C_VEL
LIN {X 0,Y 414.05,Z 622.063,A -85,B 0,C 180,E1 -10697.751,E2 -10697.751} C_VEL
LIN {X 0,Y 413.513,Z 629.805,A -85,B 0,C 180,E1 -10698.977,E2 -10698.977} C_VEL
LIN {X 0,Y 412.835,Z 637.49,A -85,B 0,C 180,E1 -10700.471,E2 -10700.471} C_VEL
LIN {X 0,Y 412.365,Z 643.245,A -85,B 0,C 180,E1 -10701.867,E2 -10701.867} C_VEL
LIN {X 0,Y 412.086,Z 647.516,A -85,B 0,C 180,E1 -10703.144,E2 -10703.144} C_VEL
LIN {X 0,Y 411.622,Z 651.409,A -85,B 0,C 180,E1 -10704.612,E2 -10704.612} C_VEL
LIN {X 0,Y 411.327,Z 654.277,A -85,B 0,C 180,E1 -10706.081,E2 -10706.081} C_VEL
LIN {X 0,Y 411.341,Z 655.63,A -85,B 0,C 180,E1 -10707.062,E2 -10707.062} C_VEL
LIN {X 0,Y 411.181,Z 656.615,A -85,B 0,C 180,E1 -10708.041,E2 -10708.041} C_VEL
LIN {X 0,Y 411.236,Z 657.406,A -85,B 0,C 180,E1 -10709.91,E2 -10709.91} C_VEL
LIN {X 0,Y 410.586,Z 657.53,A -85,B 0,C 180,E1 -10710.729,E2 -10710.729} C_VEL
LIN {X 0,Y 407.725,Z 657.299,A -85,B 0,C 180,E1 -10712.061,E2 -10712.061} C_VEL
LIN {X 0,Y 404.908,Z 656.219,A -85,B 0,C 180,E1 -10713.398,E2 -10713.398} C_VEL
LIN {X 0,Y 404.336,Z 655.01,A -85,B 0,C 180,E1 -10714.216,E2 -10714.216} C_VEL
LIN {X 0,Y 404.666,Z 651.444,A -85,B 0,C 180,E1 -10715.981,E2 -10715.981} C_VEL
LIN {X 0,Y 405.204,Z 647.259,A -85,B 0,C 180,E1 -10717.474,E2 -10717.474} C_VEL
LIN {X 0,Y 405.646,Z 640.968,A -85,B 0,C 180,E1 -10719.222,E2 -10719.222} C_VEL
LIN {X 0,Y 406.366,Z 634.005,A -85,B 0,C 180,E1 -10720.714,E2 -10720.714} C_VEL
LIN {X 0,Y 407.065,Z 625.341,A -85,B 0,C 180,E1 -10722.21,E2 -10722.21} C_VEL
LIN {X 0,Y 407.71,Z 616.437,A -85,B 0,C 180,E1 -10723.456,E2 -10723.456} C_VEL
LIN {X 0,Y 408.441,Z 606.54,A -85,B 0,C 180,E1 -10724.575,E2 -10724.575} C_VEL
LIN {X 0,Y 409.185,Z 595.39,A -85,B 0,C 180,E1 -10725.577,E2 -10725.577} C_VEL
LIN {X 0,Y 409.639,Z 585.851,A -85,B 0,C 180,E1 -10726.266,E2 -10726.266} C_VEL
LIN {X 0,Y 409.992,Z 573.81,A -85,B 0,C 180,E1 -10726.942,E2 -10726.942} C_VEL
LIN {X 0,Y 410.182,Z 561.114,A -85,B 0,C 180,E1 -10727.448,E2 -10727.448} C_VEL
LIN {X 0,Y 410.191,Z 547.599,A -85,B 0,C 180,E1 -10727.769,E2 -10727.769} C_VEL
LIN {X 0,Y 410.737,Z 490.961,A -85,B 0,C 180,E1 -10728.771,E2 -10728.771} C_VEL
LIN {X 0,Y 404.404,Z 475.006,A -85,B 0,C 180,E1 -10729.42,E2 -10729.42} C_VEL
LIN {X 0,Y 404.228,Z 474.204,A -85,B 0,C 180,E1 -10729.625,E2 -10729.625} C_VEL
LIN {X 0,Y 404.17,Z 474.132,A -85,B 0,C 180,E1 -10733.574,E2 -10733.574} C_VEL
LIN {X 0,Y 404.184,Z 474.125,A -85,B 0,C 180,E1 -10735.766,E2 -10735.766} C_VEL
LIN {X 0,Y 404.195,Z 474.113,A -85,B 0,C 180,E1 -10737.999,E2 -10737.999} C_VEL
LIN {X 0,Y 404.139,Z 474.138,A -85,B 0,C 180,E1 -10741.557,E2 -10741.557} C_VEL
LIN {X 0,Y 404.184,Z 474.139,A -85,B 0,C 180,E1 -10745.015,E2 -10745.015} C_VEL
LIN {X 0,Y 404.156,Z 474.139,A -85,B 0,C 180,E1 -10748.756,E2 -10748.756} C_VEL
LIN {X 0,Y 404.121,Z 474.134,A -85,B 0,C 180,E1 -10751.599,E2 -10751.599} C_VEL
LIN {X 0,Y 404.145,Z 474.136,A -85,B 0,C 180,E1 -10754.522,E2 -10754.522} C_VEL
LIN {X 0,Y 404.132,Z 474.141,A -85,B 0,C 180,E1 -10757.295,E2 -10757.295} C_VEL
LIN {X 0,Y 404.164,Z 474.11,A -85,B 0,C 180,E1 -10759.955,E2 -10759.955} C_VEL
LIN {X 0,Y 404.134,Z 474.142,A -85,B 0,C 180,E1 -10763.124,E2 -10763.124} C_VEL
LIN {X 0,Y 404.139,Z 474.136,A -85,B 0,C 180,E1 -10766.187,E2 -10766.187} C_VEL
LIN {X 0,Y 404.147,Z 474.11,A -85,B 0,C 180,E1 -10769.715,E2 -10769.715} C_VEL
LIN {X 0,Y 404.189,Z 474.133,A -85,B 0,C 180,E1 -10773.122,E2 -10773.122} C_VEL
LIN {X 0,Y 404.17,Z 474.14,A -85,B 0,C 180,E1 -10775.334,E2 -10775.334} C_VEL
LIN {X 0,Y 404.131,Z 474.135,A -85,B 0,C 180,E1 -10778.58,E2 -10778.58} C_VEL
LIN {X 0,Y 404.202,Z 474.132,A -85,B 0,C 180,E1 -10781.761,E2 -10781.761} C_VEL
LIN {X 0,Y 404.198,Z 474.126,A -85,B 0,C 180,E1 -10784.882,E2 -10784.882} C_VEL
LIN {X 0,Y 404.249,Z 474.126,A -85,B 0,C 180,E1 -10787.958,E2 -10787.958} C_VEL
LIN {X 0,Y 404.425,Z 474.101,A -85,B 0,C 180,E1 -10792.099,E2 -10792.099} C_VEL
LIN {X 0,Y 404.415,Z 474.105,A -85,B 0,C 180,E1 -10794.015,E2 -10794.015} C_VEL
LIN {X 0,Y 404.474,Z 474.092,A -85,B 0,C 180,E1 -10798.008,E2 -10798.008} C_VEL
LIN {X 0,Y 404.604,Z 474.082,A -85,B 0,C 180,E1 -10800,E2 -10800} C_VEL
LIN {X 0,Y 404.416,Z 474.103,A -85,B 0,C 180,E1 -10802.988,E2 -10802.988} C_VEL
LIN {X 0,Y 404.429,Z 474.104,A -85,B 0,C 180,E1 -10805.985,E2 -10805.985} C_VEL
LIN {X 0,Y 404.283,Z 474.123,A -85,B 0,C 180,E1 -10809.001,E2 -10809.001} C_VEL
LIN {X 0,Y 404.248,Z 474.125,A -85,B 0,C 180,E1 -10812.042,E2 -10812.042} C_VEL
LIN {X 0,Y 404.197,Z 474.136,A -85,B 0,C 180,E1 -10815.118,E2 -10815.118} C_VEL
LIN {X 0,Y 404.202,Z 474.112,A -85,B 0,C 180,E1 -10818.238,E2 -10818.238} C_VEL
LIN {X 0,Y 404.131,Z 474.138,A -85,B 0,C 180,E1 -10821.42,E2 -10821.42} C_VEL
LIN {X 0,Y 404.169,Z 474.134,A -85,B 0,C 180,E1 -10824.666,E2 -10824.666} C_VEL
LIN {X 0,Y 404.191,Z 474.129,A -85,B 0,C 180,E1 -10828,E2 -10828} C_VEL
LIN {X 0,Y 404.144,Z 474.143,A -85,B 0,C 180,E1 -10831.446,E2 -10831.446} C_VEL
LIN {X 0,Y 404.18,Z 474.135,A -85,B 0,C 180,E1 -10835.017,E2 -10835.017} C_VEL
LIN {X 0,Y 404.154,Z 474.134,A -85,B 0,C 180,E1 -10838.757,E2 -10838.757} C_VEL
LIN {X 0,Y 404.119,Z 474.143,A -85,B 0,C 180,E1 -10841.601,E2 -10841.601} C_VEL
LIN {X 0,Y 404.149,Z 474.12,A -85,B 0,C 180,E1 -10844.524,E2 -10844.524} C_VEL
LIN {X 0,Y 404.208,Z 474.137,A -85,B 0,C 180,E1 -10847.306,E2 -10847.306} C_VEL
LIN {X 0,Y 404.166,Z 474.126,A -85,B 0,C 180,E1 -10849.956,E2 -10849.956} C_VEL
LIN {X 0,Y 404.138,Z 474.134,A -85,B 0,C 180,E1 -10853.125,E2 -10853.125} C_VEL
LIN {X 0,Y 404.143,Z 474.135,A -85,B 0,C 180,E1 -10856.189,E2 -10856.189} C_VEL
LIN {X 0,Y 404.207,Z 474.405,A -85,B 0,C 180,E1 -10857.052,E2 -10857.052} C_VEL
LIN {X 0,Y 407.753,Z 489.354,A -85,B 0,C 180,E1 -10859.797,E2 -10859.797} C_VEL
LIN {X 0,Y 409.395,Z 497.826,A -85,B 0,C 180,E1 -10861.272,E2 -10861.272} C_VEL
LIN {X 0,Y 408.037,Z 516.755,A -85,B 0,C 180,E1 -10864.228,E2 -10864.228} C_VEL
LIN {X 0,Y 406.551,Z 538.789,A -85,B 0,C 180,E1 -10867.648,E2 -10867.648} C_VEL
LIN {X 0,Y 405.609,Z 555.21,A -85,B 0,C 180,E1 -10870.187,E2 -10870.187} C_VEL
LIN {X 0,Y 408.737,Z 583.466,A -85,B 0,C 180,E1 -10870.88,E2 -10870.88} C_VEL
LIN {X 0,Y 409.843,Z 595.452,A -85,B 0,C 180,E1 -10871.147,E2 -10871.147} C_VEL
LIN {X 0,Y 409.015,Z 665.943,A -85,B 0,C 180,E1 -10872.404,E2 -10872.404} C_VEL
LIN {X 0,Y 408.39,Z 679.234,A -85,B 0,C 180,E1 -10872.828,E2 -10872.828} C_VEL
LIN {X 0,Y 407.648,Z 691.453,A -85,B 0,C 180,E1 -10873.409,E2 -10873.409} C_VEL
LIN {X 0,Y 406.895,Z 702.114,A -85,B 0,C 180,E1 -10874.086,E2 -10874.086} C_VEL
LIN {X 0,Y 406.009,Z 712.89,A -85,B 0,C 180,E1 -10874.951,E2 -10874.951} C_VEL
LIN {X 0,Y 405.142,Z 724.215,A -85,B 0,C 180,E1 -10876.105,E2 -10876.105} C_VEL
LIN {X 0,Y 404.682,Z 733.018,A -85,B 0,C 180,E1 -10877.208,E2 -10877.208} C_VEL
LIN {X 0,Y 404.027,Z 741.346,A -85,B 0,C 180,E1 -10878.461,E2 -10878.461} C_VEL
LIN {X 0,Y 403.557,Z 749.559,A -85,B 0,C 180,E1 -10879.971,E2 -10879.971} C_VEL
LIN {X 0,Y 403.369,Z 756.188,A -85,B 0,C 180,E1 -10881.484,E2 -10881.484} C_VEL
LIN {X 0,Y 403.345,Z 762.404,A -85,B 0,C 180,E1 -10883.309,E2 -10883.309} C_VEL
LIN {X 0,Y 403.475,Z 766.717,A -85,B 0,C 180,E1 -10885.004,E2 -10885.004} C_VEL
LIN {X 0,Y 403.595,Z 768.663,A -85,B 0,C 180,E1 -10886.006,E2 -10886.006} C_VEL
LIN {X 0,Y 403.56,Z 770.106,A -85,B 0,C 180,E1 -10887.005,E2 -10887.005} C_VEL
LIN {X 0,Y 403.853,Z 771.81,A -85,B 0,C 180,E1 -10889.003,E2 -10889.003} C_VEL
LIN {X 0,Y 403.879,Z 772.037,A -85,B 0,C 180,E1 -10890,E2 -10890} C_VEL
LIN {X 0,Y 403.853,Z 771.809,A -85,B 0,C 180,E1 -10890.997,E2 -10890.997} C_VEL
LIN {X 0,Y 403.56,Z 770.105,A -85,B 0,C 180,E1 -10892.995,E2 -10892.995} C_VEL
LIN {X 0,Y 403.595,Z 768.66,A -85,B 0,C 180,E1 -10893.994,E2 -10893.994} C_VEL
LIN {X 0,Y 403.389,Z 765.587,A -85,B 0,C 180,E1 -10895.499,E2 -10895.499} C_VEL
LIN {X 0,Y 403.351,Z 761.464,A -85,B 0,C 180,E1 -10897.006,E2 -10897.006} C_VEL
LIN {X 0,Y 403.382,Z 755.139,A -85,B 0,C 180,E1 -10898.769,E2 -10898.769} C_VEL
LIN {X 0,Y 403.602,Z 748.267,A -85,B 0,C 180,E1 -10900.281,E2 -10900.281} C_VEL
LIN {X 0,Y 404.102,Z 739.791,A -85,B 0,C 180,E1 -10901.791,E2 -10901.791} C_VEL
LIN {X 0,Y 404.768,Z 731.138,A -85,B 0,C 180,E1 -10903.045,E2 -10903.045} C_VEL
LIN {X 0,Y 405.377,Z 721.655,A -85,B 0,C 180,E1 -10904.175,E2 -10904.175} C_VEL
LIN {X 0,Y 406.236,Z 709.948,A -85,B 0,C 180,E1 -10905.297,E2 -10905.297} C_VEL
LIN {X 0,Y 407.129,Z 698.463,A -85,B 0,C 180,E1 -10906.162,E2 -10906.162} C_VEL
LIN {X 0,Y 407.957,Z 686.695,A -85,B 0,C 180,E1 -10906.836,E2 -10906.836} C_VEL
LIN {X 0,Y 408.717,Z 673.171,A -85,B 0,C 180,E1 -10907.383,E2 -10907.383} C_VEL
LIN {X 0,Y 409.112,Z 659.77,A -85,B 0,C 180,E1 -10907.721,E2 -10907.721} C_VEL
LIN {X 0,Y 409.746,Z 593.354,A -85,B 0,C 180,E1 -10908.888,E2 -10908.888} C_VEL
LIN {X 0,Y 405.592,Z 555.548,A -85,B 0,C 180,E1 -10909.781,E2 -10909.781} C_VEL
LIN {X 0,Y 406.095,Z 546.482,A -85,B 0,C 180,E1 -10911.147,E2 -10911.147} C_VEL
LIN {X 0,Y 407.408,Z 525.165,A -85,B 0,C 180,E1 -10914.457,E2 -10914.457} C_VEL
LIN {X 0,Y 408.894,Z 504.641,A -85,B 0,C 180,E1 -10917.649,E2 -10917.649} C_VEL
LIN {X 0,Y 409.395,Z 497.767,A -85,B 0,C 180,E1 -10918.728,E2 -10918.728} C_VEL
LIN {X 0,Y 407.743,Z 489.336,A -85,B 0,C 180,E1 -10920.195,E2 -10920.195} C_VEL
LIN {X 0,Y 404.202,Z 474.26,A -85,B 0,C 180,E1 -10922.982,E2 -10922.982} C_VEL
LIN {X 0,Y 404.141,Z 474.132,A -85,B 0,C 180,E1 -10926.245,E2 -10926.245} C_VEL
LIN {X 0,Y 404.16,Z 474.139,A -85,B 0,C 180,E1 -10928.755,E2 -10928.755} C_VEL
LIN {X 0,Y 404.188,Z 474.13,A -85,B 0,C 180,E1 -10931.61,E2 -10931.61} C_VEL
LIN {X 0,Y 404.189,Z 474.125,A -85,B 0,C 180,E1 -10934.528,E2 -10934.528} C_VEL
LIN {X 0,Y 404.131,Z 474.131,A -85,B 0,C 180,E1 -10937.295,E2 -10937.295} C_VEL
LIN {X 0,Y 404.164,Z 474.142,A -85,B 0,C 180,E1 -10939.955,E2 -10939.955} C_VEL
LIN {X 0,Y 404.134,Z 474.141,A -85,B 0,C 180,E1 -10943.124,E2 -10943.124} C_VEL
LIN {X 0,Y 404.139,Z 474.135,A -85,B 0,C 180,E1 -10946.187,E2 -10946.187} C_VEL
LIN {X 0,Y 404.157,Z 474.14,A -85,B 0,C 180,E1 -10949.716,E2 -10949.716} C_VEL
LIN {X 0,Y 404.188,Z 474.119,A -85,B 0,C 180,E1 -10953.122,E2 -10953.122} C_VEL
LIN {X 0,Y 404.169,Z 474.134,A -85,B 0,C 180,E1 -10955.334,E2 -10955.334} C_VEL
LIN {X 0,Y 404.131,Z 474.138,A -85,B 0,C 180,E1 -10958.58,E2 -10958.58} C_VEL
LIN {X 0,Y 404.202,Z 474.113,A -85,B 0,C 180,E1 -10961.762,E2 -10961.762} C_VEL
LIN {X 0,Y 404.197,Z 474.136,A -85,B 0,C 180,E1 -10964.882,E2 -10964.882} C_VEL
LIN {X 0,Y 404.248,Z 474.124,A -85,B 0,C 180,E1 -10967.958,E2 -10967.958} C_VEL
LIN {X 0,Y 404.396,Z 474.111,A -85,B 0,C 180,E1 -10972.128,E2 -10972.128} C_VEL
LIN {X 0,Y 404.429,Z 474.104,A -85,B 0,C 180,E1 -10974.015,E2 -10974.015} C_VEL
LIN {X 0,Y 404.474,Z 474.097,A -85,B 0,C 180,E1 -10978.009,E2 -10978.009} C_VEL
LIN {X 0,Y 404.604,Z 474.083,A -85,B 0,C 180,E1 -10980,E2 -10980} C_VEL
LIN {X 0,Y 404.416,Z 474.099,A -85,B 0,C 180,E1 -10982.988,E2 -10982.988} C_VEL
LIN {X 0,Y 404.394,Z 474.107,A -85,B 0,C 180,E1 -10986.612,E2 -10986.612} C_VEL
LIN {X 0,Y 404.283,Z 474.113,A -85,B 0,C 180,E1 -10989.001,E2 -10989.001} C_VEL
LIN {X 0,Y 404.249,Z 474.126,A -85,B 0,C 180,E1 -10992.042,E2 -10992.042} C_VEL
LIN {X 0,Y 404.198,Z 474.126,A -85,B 0,C 180,E1 -10995.118,E2 -10995.118} C_VEL
LIN {X 0,Y 404.202,Z 474.131,A -85,B 0,C 180,E1 -10998.239,E2 -10998.239} C_VEL
LIN {X 0,Y 404.131,Z 474.135,A -85,B 0,C 180,E1 -11001.42,E2 -11001.42} C_VEL
LIN {X 0,Y 404.17,Z 474.139,A -85,B 0,C 180,E1 -11004.666,E2 -11004.666} C_VEL
LIN {X 0,Y 404.192,Z 474.126,A -85,B 0,C 180,E1 -11008,E2 -11008} C_VEL
LIN {X 0,Y 404.136,Z 474.116,A -85,B 0,C 180,E1 -11011.56,E2 -11011.56} C_VEL
LIN {X 0,Y 404.18,Z 474.141,A -85,B 0,C 180,E1 -11015.017,E2 -11015.017} C_VEL
LIN {X 0,Y 404.147,Z 474.124,A -85,B 0,C 180,E1 -11018.758,E2 -11018.758} C_VEL
LIN {X 0,Y 404.119,Z 474.136,A -85,B 0,C 180,E1 -11021.601,E2 -11021.601} C_VEL
LIN {X 0,Y 404.143,Z 474.143,A -85,B 0,C 180,E1 -11024.523,E2 -11024.523} C_VEL
LIN {X 0,Y 404.136,Z 474.127,A -85,B 0,C 180,E1 -11027.297,E2 -11027.297} C_VEL
LIN {X 0,Y 404.166,Z 474.138,A -85,B 0,C 180,E1 -11029.956,E2 -11029.956} C_VEL
LIN {X 0,Y 404.138,Z 474.122,A -85,B 0,C 180,E1 -11033.125,E2 -11033.125} C_VEL
LIN {X 0,Y 404.144,Z 474.099,A -85,B 0,C 180,E1 -11036.189,E2 -11036.189} C_VEL
LIN {X 0,Y 404.145,Z 474.144,A -85,B 0,C 180,E1 -11039.716,E2 -11039.716} C_VEL
LIN {X 0,Y 404.195,Z 474.109,A -85,B 0,C 180,E1 -11043.124,E2 -11043.124} C_VEL
LIN {X 0,Y 404.179,Z 474.141,A -85,B 0,C 180,E1 -11045.335,E2 -11045.335} C_VEL
LIN {X 0,Y 404.14,Z 474.128,A -85,B 0,C 180,E1 -11048.581,E2 -11048.581} C_VEL
LIN {X 0,Y 404.273,Z 474.299,A -85,B 0,C 180,E1 -11050.545,E2 -11050.545} C_VEL
LIN {X 0,Y 404.498,Z 475.308,A -85,B 0,C 180,E1 -11050.707,E2 -11050.707} C_VEL
LIN {X 0,Y 410.72,Z 490.921,A -85,B 0,C 180,E1 -11051.327,E2 -11051.327} C_VEL
LIN {X 0,Y 410.245,Z 555.348,A -85,B 0,C 180,E1 -11052.491,E2 -11052.491} C_VEL
LIN {X 0,Y 410.074,Z 568.775,A -85,B 0,C 180,E1 -11052.933,E2 -11052.933} C_VEL
LIN {X 0,Y 409.752,Z 581.485,A -85,B 0,C 180,E1 -11053.561,E2 -11053.561} C_VEL
LIN {X 0,Y 409.293,Z 593.108,A -85,B 0,C 180,E1 -11054.339,E2 -11054.339} C_VEL
LIN {X 0,Y 408.537,Z 604.29,A -85,B 0,C 180,E1 -11055.301,E2 -11055.301} C_VEL
LIN {X 0,Y 407.825,Z 614.625,A -85,B 0,C 180,E1 -11056.421,E2 -11056.421} C_VEL
LIN {X 0,Y 407.184,Z 623.054,A -85,B 0,C 180,E1 -11057.541,E2 -11057.541} C_VEL
LIN {X 0,Y 406.617,Z 630.795,A -85,B 0,C 180,E1 -11058.788,E2 -11058.788} C_VEL
LIN {X 0,Y 405.905,Z 638.48,A -85,B 0,C 180,E1 -11060.306,E2 -11060.306} C_VEL
LIN {X 0,Y 405.409,Z 644.234,A -85,B 0,C 180,E1 -11061.726,E2 -11061.726} C_VEL
LIN {X 0,Y 405.11,Z 648.505,A -85,B 0,C 180,E1 -11063.025,E2 -11063.025} C_VEL
LIN {X 0,Y 404.624,Z 652.399,A -85,B 0,C 180,E1 -11064.518,E2 -11064.518} C_VEL
LIN {X 0,Y 404.313,Z 655.266,A -85,B 0,C 180,E1 -11066.013,E2 -11066.013} C_VEL
LIN {X 0,Y 404.323,Z 656.619,A -85,B 0,C 180,E1 -11067.011,E2 -11067.011} C_VEL
LIN {X 0,Y 404.159,Z 657.603,A -85,B 0,C 180,E1 -11068.007,E2 -11068.007} C_VEL
LIN {X 0,Y 404.212,Z 658.394,A -85,B 0,C 180,E1 -11069.91,E2 -11069.91} C_VEL
LIN {X 0,Y 404.232,Z 658.231,A -85,B 0,C 180,E1 -11070.996,E2 -11070.996} C_VEL
LIN {X 0,Y 404.159,Z 657.677,A -85,B 0,C 180,E1 -11071.993,E2 -11071.993} C_VEL
LIN {X 0,Y 404.321,Z 656.722,A -85,B 0,C 180,E1 -11072.989,E2 -11072.989} C_VEL
LIN {X 0,Y 404.336,Z 655.01,A -85,B 0,C 180,E1 -11074.216,E2 -11074.216} C_VEL
LIN {X 0,Y 403.833,Z 653.67,A -85,B 0,C 180,E1 -11075.026,E2 -11075.026} C_VEL
LIN {X 0,Y 401.343,Z 651.172,A -85,B 0,C 180,E1 -11076.346,E2 -11076.346} C_VEL
LIN {X 0,Y 399.249,Z 648.702,A -85,B 0,C 180,E1 -11077.39,E2 -11077.39} C_VEL
LIN {X 0,Y 398.43,Z 646.424,A -85,B 0,C 180,E1 -11078.169,E2 -11078.169} C_VEL
LIN {X 0,Y 398.408,Z 645.55,A -85,B 0,C 180,E1 -11078.425,E2 -11078.425} C_VEL
LIN {X 0,Y 398.94,Z 639.785,A -85,B 0,C 180,E1 -11079.89,E2 -11079.89} C_VEL
LIN {X 0,Y 399.721,Z 632.336,A -85,B 0,C 180,E1 -11081.408,E2 -11081.408} C_VEL
LIN {X 0,Y 400.303,Z 624.715,A -85,B 0,C 180,E1 -11082.677,E2 -11082.677} C_VEL
LIN {X 0,Y 401.057,Z 614.334,A -85,B 0,C 180,E1 -11084.072,E2 -11084.072} C_VEL
LIN {X 0,Y 401.891,Z 603.711,A -85,B 0,C 180,E1 -11085.207,E2 -11085.207} C_VEL
LIN {X 0,Y 402.578,Z 592.877,A -85,B 0,C 180,E1 -11086.123,E2 -11086.123} C_VEL
LIN {X 0,Y 403.174,Z 580.159,A -85,B 0,C 180,E1 -11086.95,E2 -11086.95} C_VEL
LIN {X 0,Y 403.454,Z 568.304,A -85,B 0,C 180,E1 -11087.519,E2 -11087.519} C_VEL
LIN {X 0,Y 403.556,Z 556.415,A -85,B 0,C 180,E1 -11087.907,E2 -11087.907} C_VEL
LIN {X 0,Y 403.779,Z 518.889,A -85,B 0,C 180,E1 -11088.608,E2 -11088.608} C_VEL
LIN {X 0,Y 404.043,Z 492.638,A -85,B 0,C 180,E1 -11089.08,E2 -11089.08} C_VEL
LIN {X 0,Y 397.362,Z 476.031,A -85,B 0,C 180,E1 -11089.768,E2 -11089.768} C_VEL
LIN {X 0,Y 397.18,Z 475.115,A -85,B 0,C 180,E1 -11089.96,E2 -11089.96} C_VEL
LIN {X 0,Y 397.134,Z 475.016,A -85,B 0,C 180,E1 -11094.018,E2 -11094.018} C_VEL
LIN {X 0,Y 397.194,Z 474.979,A -85,B 0,C 180,E1 -11097.389,E2 -11097.389} C_VEL
LIN {X 0,Y 397.079,Z 475.025,A -85,B 0,C 180,E1 -11100.882,E2 -11100.882} C_VEL
LIN {X 0,Y 397.125,Z 475.017,A -85,B 0,C 180,E1 -11104.492,E2 -11104.492} C_VEL
LIN {X 0,Y 397.104,Z 475.014,A -85,B 0,C 180,E1 -11108.274,E2 -11108.274} C_VEL
LIN {X 0,Y 397.086,Z 475.018,A -85,B 0,C 180,E1 -11110.908,E2 -11110.908} C_VEL
LIN {X 0,Y 397.1,Z 475.01,A -85,B 0,C 180,E1 -11113.647,E2 -11113.647} C_VEL
LIN {X 0,Y 397.098,Z 475.021,A -85,B 0,C 180,E1 -11116.52,E2 -11116.52} C_VEL
LIN {X 0,Y 397.108,Z 474.989,A -85,B 0,C 180,E1 -11120.422,E2 -11120.422} C_VEL
LIN {X 0,Y 397.104,Z 475.017,A -85,B 0,C 180,E1 -11124.265,E2 -11124.265} C_VEL
LIN {X 0,Y 397.109,Z 475.01,A -85,B 0,C 180,E1 -11126.726,E2 -11126.726} C_VEL
LIN {X 0,Y 397.127,Z 474.988,A -85,B 0,C 180,E1 -11130.296,E2 -11130.296} C_VEL
LIN {X 0,Y 397.188,Z 475,A -85,B 0,C 180,E1 -11132.609,E2 -11132.609} C_VEL
LIN {X 0,Y 397.126,Z 475.012,A -85,B 0,C 180,E1 -11135.981,E2 -11135.981} C_VEL
LIN {X 0,Y 397.131,Z 475.016,A -85,B 0,C 180,E1 -11139.704,E2 -11139.704} C_VEL
LIN {X 0,Y 397.174,Z 475.007,A -85,B 0,C 180,E1 -11142.844,E2 -11142.844} C_VEL
LIN {X 0,Y 397.22,Z 475.003,A -85,B 0,C 180,E1 -11146.702,E2 -11146.702} C_VEL
LIN {X 0,Y 397.21,Z 474.993,A -85,B 0,C 180,E1 -11149.809,E2 -11149.809} C_VEL
LIN {X 0,Y 397.355,Z 474.983,A -85,B 0,C 180,E1 -11152.888,E2 -11152.888} C_VEL
LIN {X 0,Y 397.248,Z 474.999,A -85,B 0,C 180,E1 -11154.925,E2 -11154.925} C_VEL
LIN {X 0,Y 397.443,Z 474.967,A -85,B 0,C 180,E1 -11157.973,E2 -11157.973} C_VEL
LIN {X 0,Y 397.574,Z 474.957,A -85,B 0,C 180,E1 -11160,E2 -11160} C_VEL
LIN {X 0,Y 397.374,Z 474.98,A -85,B 0,C 180,E1 -11163.041,E2 -11163.041} C_VEL
LIN {X 0,Y 397.377,Z 474.982,A -85,B 0,C 180,E1 -11166.091,E2 -11166.091} C_VEL
LIN {X 0,Y 397.245,Z 475.001,A -85,B 0,C 180,E1 -11169.162,E2 -11169.162} C_VEL
LIN {X 0,Y 397.211,Z 475,A -85,B 0,C 180,E1 -11172.258,E2 -11172.258} C_VEL
LIN {X 0,Y 397.17,Z 475.013,A -85,B 0,C 180,E1 -11175.392,E2 -11175.392} C_VEL
LIN {X 0,Y 397.154,Z 474.988,A -85,B 0,C 180,E1 -11178.574,E2 -11178.574} C_VEL
LIN {X 0,Y 397.089,Z 475.021,A -85,B 0,C 180,E1 -11181.819,E2 -11181.819} C_VEL
LIN {X 0,Y 397.149,Z 475.011,A -85,B 0,C 180,E1 -11185.132,E2 -11185.132} C_VEL
LIN {X 0,Y 397.157,Z 475.001,A -85,B 0,C 180,E1 -11187.777,E2 -11187.777} C_VEL
LIN {X 0,Y 397.085,Z 475.02,A -85,B 0,C 180,E1 -11190.882,E2 -11190.882} C_VEL
LIN {X 0,Y 397.12,Z 475.014,A -85,B 0,C 180,E1 -11194.494,E2 -11194.494} C_VEL
LIN {X 0,Y 397.101,Z 475.012,A -85,B 0,C 180,E1 -11198.275,E2 -11198.275} C_VEL
LIN {X 0,Y 397.085,Z 475.021,A -85,B 0,C 180,E1 -11200.909,E2 -11200.909} C_VEL
LIN {X 0,Y 397.098,Z 474.996,A -85,B 0,C 180,E1 -11203.649,E2 -11203.649} C_VEL
LIN {X 0,Y 397.161,Z 475.013,A -85,B 0,C 180,E1 -11206.512,E2 -11206.512} C_VEL
LIN {X 0,Y 397.12,Z 475.002,A -85,B 0,C 180,E1 -11209.552,E2 -11209.552} C_VEL
LIN {X 0,Y 397.096,Z 475.014,A -85,B 0,C 180,E1 -11212.791,E2 -11212.791} C_VEL
LIN {X 0,Y 397.117,Z 475.009,A -85,B 0,C 180,E1 -11216.283,E2 -11216.283} C_VEL
LIN {X 0,Y 397.159,Z 475.266,A -85,B 0,C 180,E1 -11216.704,E2 -11216.704} C_VEL
LIN {X 0,Y 401.005,Z 491.483,A -85,B 0,C 180,E1 -11219.744,E2 -11219.744} C_VEL
LIN {X 0,Y 402.472,Z 498.903,A -85,B 0,C 180,E1 -11221.063,E2 -11221.063} C_VEL
LIN {X 0,Y 401.23,Z 516.112,A -85,B 0,C 180,E1 -11223.808,E2 -11223.808} C_VEL
LIN {X 0,Y 399.58,Z 539.482,A -85,B 0,C 180,E1 -11227.509,E2 -11227.509} C_VEL
LIN {X 0,Y 398.697,Z 554.191,A -85,B 0,C 180,E1 -11229.829,E2 -11229.829} C_VEL
LIN {X 0,Y 401.956,Z 583.551,A -85,B 0,C 180,E1 -11230.565,E2 -11230.565} C_VEL
LIN {X 0,Y 403.114,Z 596.591,A -85,B 0,C 180,E1 -11230.859,E2 -11230.859} C_VEL
LIN {X 0,Y 402.246,Z 664.956,A -85,B 0,C 180,E1 -11232.098,E2 -11232.098} C_VEL
LIN {X 0,Y 401.614,Z 678.245,A -85,B 0,C 180,E1 -11232.529,E2 -11232.529} C_VEL
LIN {X 0,Y 400.732,Z 691.584,A -85,B 0,C 180,E1 -11233.18,E2 -11233.18} C_VEL
LIN {X 0,Y 399.888,Z 702.819,A -85,B 0,C 180,E1 -11233.931,E2 -11233.931} C_VEL
LIN {X 0,Y 398.886,Z 714.529,A -85,B 0,C 180,E1 -11234.937,E2 -11234.937} C_VEL
LIN {X 0,Y 398.035,Z 725.174,A -85,B 0,C 180,E1 -11236.087,E2 -11236.087} C_VEL
LIN {X 0,Y 397.537,Z 733.827,A -85,B 0,C 180,E1 -11237.233,E2 -11237.233} C_VEL
LIN {X 0,Y 396.913,Z 741.862,A -85,B 0,C 180,E1 -11238.51,E2 -11238.51} C_VEL
LIN {X 0,Y 396.476,Z 749.753,A -85,B 0,C 180,E1 -11240.048,E2 -11240.048} C_VEL
LIN {X 0,Y 396.288,Z 757.068,A -85,B 0,C 180,E1 -11241.844,E2 -11241.844} C_VEL
LIN {X 0,Y 396.293,Z 761.667,A -85,B 0,C 180,E1 -11243.279,E2 -11243.279} C_VEL
LIN {X 0,Y 396.39,Z 765.717,A -85,B 0,C 180,E1 -11244.914,E2 -11244.914} C_VEL
LIN {X 0,Y 396.535,Z 767.668,A -85,B 0,C 180,E1 -11245.935,E2 -11245.935} C_VEL
LIN {X 0,Y 396.515,Z 769.115,A -85,B 0,C 180,E1 -11246.952,E2 -11246.952} C_VEL
LIN {X 0,Y 396.824,Z 770.822,A -85,B 0,C 180,E1 -11248.985,E2 -11248.985} C_VEL
LIN {X 0,Y 396.856,Z 771.05,A -85,B 0,C 180,E1 -11250,E2 -11250} C_VEL
LIN {X 0,Y 396.824,Z 770.82,A -85,B 0,C 180,E1 -11251.015,E2 -11251.015} C_VEL
LIN {X 0,Y 396.516,Z 769.113,A -85,B 0,C 180,E1 -11253.048,E2 -11253.048} C_VEL
LIN {X 0,Y 396.535,Z 767.664,A -85,B 0,C 180,E1 -11254.065,E2 -11254.065} C_VEL
LIN {X 0,Y 396.32,Z 764.588,A -85,B 0,C 180,E1 -11255.597,E2 -11255.597} C_VEL
LIN {X 0,Y 396.287,Z 760.462,A -85,B 0,C 180,E1 -11257.131,E2 -11257.131} C_VEL
LIN {X 0,Y 396.323,Z 754.133,A -85,B 0,C 180,E1 -11258.926,E2 -11258.926} C_VEL
LIN {X 0,Y 396.568,Z 747.26,A -85,B 0,C 180,E1 -11260.466,E2 -11260.466} C_VEL
LIN {X 0,Y 397.061,Z 738.777,A -85,B 0,C 180,E1 -11262.003,E2 -11262.003} C_VEL
LIN {X 0,Y 397.765,Z 730.124,A -85,B 0,C 180,E1 -11263.279,E2 -11263.279} C_VEL
LIN {X 0,Y 398.461,Z 720.649,A -85,B 0,C 180,E1 -11264.426,E2 -11264.426} C_VEL
LIN {X 0,Y 399.226,Z 710.381,A -85,B 0,C 180,E1 -11265.442,E2 -11265.442} C_VEL
LIN {X 0,Y 400.158,Z 699.241,A -85,B 0,C 180,E1 -11266.32,E2 -11266.32} C_VEL
LIN {X 0,Y 401.077,Z 686.922,A -85,B 0,C 180,E1 -11267.068,E2 -11267.068} C_VEL
LIN {X 0,Y 401.856,Z 673.998,A -85,B 0,C 180,E1 -11267.624,E2 -11267.624} C_VEL
LIN {X 0,Y 402.321,Z 660.294,A -85,B 0,C 180,E1 -11267.997,E2 -11267.997} C_VEL
LIN {X 0,Y 402.954,Z 593.553,A -85,B 0,C 180,E1 -11269.196,E2 -11269.196} C_VEL
LIN {X 0,Y 398.783,Z 555.686,A -85,B 0,C 180,E1 -11270.1,E2 -11270.1} C_VEL
LIN {X 0,Y 398.669,Z 554.118,A -85,B 0,C 180,E1 -11270.173,E2 -11270.173} C_VEL
LIN {X 0,Y 400.01,Z 532.685,A -85,B 0,C 180,E1 -11273.559,E2 -11273.559} C_VEL
LIN {X 0,Y 401.643,Z 510.576,A -85,B 0,C 180,E1 -11277.061,E2 -11277.061} C_VEL
LIN {X 0,Y 402.465,Z 498.767,A -85,B 0,C 180,E1 -11278.949,E2 -11278.949} C_VEL
LIN {X 0,Y 399.774,Z 486.034,A -85,B 0,C 180,E1 -11281.237,E2 -11281.237} C_VEL
LIN {X 0,Y 397.139,Z 475.137,A -85,B 0,C 180,E1 -11283.325,E2 -11283.325} C_VEL
LIN {X 0,Y 397.107,Z 475.011,A -85,B 0,C 180,E1 -11285.734,E2 -11285.734} C_VEL
LIN {X 0,Y 397.113,Z 475.007,A -85,B 0,C 180,E1 -11289.576,E2 -11289.576} C_VEL
LIN {X 0,Y 397.157,Z 475.013,A -85,B 0,C 180,E1 -11292.254,E2 -11292.254} C_VEL
LIN {X 0,Y 397.108,Z 475,A -85,B 0,C 180,E1 -11295.064,E2 -11295.064} C_VEL
LIN {X 0,Y 397.061,Z 475.016,A -85,B 0,C 180,E1 -11298.02,E2 -11298.02} C_VEL
LIN {X 0,Y 397.128,Z 475.009,A -85,B 0,C 180,E1 -11301.137,E2 -11301.137} C_VEL
LIN {X 0,Y 397.114,Z 475.018,A -85,B 0,C 180,E1 -11304.496,E2 -11304.496} C_VEL
LIN {X 0,Y 397.075,Z 475.015,A -85,B 0,C 180,E1 -11307.928,E2 -11307.928} C_VEL
LIN {X 0,Y 397.141,Z 475.017,A -85,B 0,C 180,E1 -11310.297,E2 -11310.297} C_VEL
LIN {X 0,Y 397.188,Z 474.993,A -85,B 0,C 180,E1 -11312.609,E2 -11312.609} C_VEL
LIN {X 0,Y 397.125,Z 475.014,A -85,B 0,C 180,E1 -11315.981,E2 -11315.981} C_VEL
LIN {X 0,Y 397.131,Z 475.004,A -85,B 0,C 180,E1 -11319.704,E2 -11319.704} C_VEL
LIN {X 0,Y 397.174,Z 475.002,A -85,B 0,C 180,E1 -11322.845,E2 -11322.845} C_VEL
LIN {X 0,Y 397.22,Z 475.003,A -85,B 0,C 180,E1 -11326.702,E2 -11326.702} C_VEL
LIN {X 0,Y 397.21,Z 474.995,A -85,B 0,C 180,E1 -11329.809,E2 -11329.809} C_VEL
LIN {X 0,Y 397.345,Z 474.988,A -85,B 0,C 180,E1 -11332.888,E2 -11332.888} C_VEL
LIN {X 0,Y 397.253,Z 474.988,A -85,B 0,C 180,E1 -11334.925,E2 -11334.925} C_VEL
LIN {X 0,Y 397.443,Z 474.973,A -85,B 0,C 180,E1 -11337.973,E2 -11337.973} C_VEL
LIN {X 0,Y 397.574,Z 474.959,A -85,B 0,C 180,E1 -11340,E2 -11340} C_VEL
LIN {X 0,Y 397.374,Z 474.976,A -85,B 0,C 180,E1 -11343.042,E2 -11343.042} C_VEL
LIN {X 0,Y 397.346,Z 474.984,A -85,B 0,C 180,E1 -11346.607,E2 -11346.607} C_VEL
LIN {X 0,Y 397.245,Z 474.988,A -85,B 0,C 180,E1 -11349.162,E2 -11349.162} C_VEL
LIN {X 0,Y 397.211,Z 475.004,A -85,B 0,C 180,E1 -11352.258,E2 -11352.258} C_VEL
LIN {X 0,Y 397.171,Z 474.999,A -85,B 0,C 180,E1 -11355.392,E2 -11355.392} C_VEL
LIN {X 0,Y 397.154,Z 475.013,A -85,B 0,C 180,E1 -11358.574,E2 -11358.574} C_VEL
LIN {X 0,Y 397.089,Z 475.011,A -85,B 0,C 180,E1 -11361.819,E2 -11361.819} C_VEL
LIN {X 0,Y 397.15,Z 475.014,A -85,B 0,C 180,E1 -11365.132,E2 -11365.132} C_VEL
LIN {X 0,Y 397.157,Z 475.002,A -85,B 0,C 180,E1 -11367.777,E2 -11367.777} C_VEL
LIN {X 0,Y 397.077,Z 474.989,A -85,B 0,C 180,E1 -11370.883,E2 -11370.883} C_VEL
LIN {X 0,Y 397.12,Z 475.013,A -85,B 0,C 180,E1 -11374.494,E2 -11374.494} C_VEL
LIN {X 0,Y 397.097,Z 475.012,A -85,B 0,C 180,E1 -11378.276,E2 -11378.276} C_VEL
LIN {X 0,Y 397.084,Z 474.999,A -85,B 0,C 180,E1 -11380.91,E2 -11380.91} C_VEL
LIN {X 0,Y 397.097,Z 475.019,A -85,B 0,C 180,E1 -11383.649,E2 -11383.649} C_VEL
LIN {X 0,Y 397.101,Z 475.008,A -85,B 0,C 180,E1 -11386.521,E2 -11386.521} C_VEL
LIN {X 0,Y 397.113,Z 475.018,A -85,B 0,C 180,E1 -11390.424,E2 -11390.424} C_VEL
LIN {X 0,Y 397.108,Z 474.98,A -85,B 0,C 180,E1 -11394.266,E2 -11394.266} C_VEL
LIN {X 0,Y 397.113,Z 474.981,A -85,B 0,C 180,E1 -11396.728,E2 -11396.728} C_VEL
LIN {X 0,Y 397.124,Z 475.018,A -85,B 0,C 180,E1 -11400.297,E2 -11400.297} C_VEL
LIN {X 0,Y 397.194,Z 474.98,A -85,B 0,C 180,E1 -11402.611,E2 -11402.611} C_VEL
LIN {X 0,Y 397.134,Z 475.015,A -85,B 0,C 180,E1 -11405.982,E2 -11405.982} C_VEL
LIN {X 0,Y 397.168,Z 475.018,A -85,B 0,C 180,E1 -11409.994,E2 -11409.994} C_VEL
LIN {X 0,Y 397.259,Z 475.517,A -85,B 0,C 180,E1 -11410.269,E2 -11410.269} C_VEL
LIN {X 0,Y 398.004,Z 477.584,A -85,B 0,C 180,E1 -11410.419,E2 -11410.419} C_VEL
LIN {X 0,Y 404.044,Z 492.564,A -85,B 0,C 180,E1 -11411.018,E2 -11411.018} C_VEL
LIN {X 0,Y 403.524,Z 556.36,A -85,B 0,C 180,E1 -11412.189,E2 -11412.189} C_VEL
LIN {X 0,Y 403.353,Z 569.775,A -85,B 0,C 180,E1 -11412.64,E2 -11412.64} C_VEL
LIN {X 0,Y 403.013,Z 582.482,A -85,B 0,C 180,E1 -11413.278,E2 -11413.278} C_VEL
LIN {X 0,Y 402.545,Z 593.703,A -85,B 0,C 180,E1 -11414.038,E2 -11414.038} C_VEL
LIN {X 0,Y 401.741,Z 605.283,A -85,B 0,C 180,E1 -11415.047,E2 -11415.047} C_VEL
LIN {X 0,Y 400.996,Z 615.617,A -85,B 0,C 180,E1 -11416.185,E2 -11416.185} C_VEL
LIN {X 0,Y 400.324,Z 624.045,A -85,B 0,C 180,E1 -11417.324,E2 -11417.324} C_VEL
LIN {X 0,Y 399.725,Z 631.786,A -85,B 0,C 180,E1 -11418.592,E2 -11418.592} C_VEL
LIN {X 0,Y 398.98,Z 639.47,A -85,B 0,C 180,E1 -11420.137,E2 -11420.137} C_VEL
LIN {X 0,Y 398.455,Z 645.224,A -85,B 0,C 180,E1 -11421.581,E2 -11421.581} C_VEL
LIN {X 0,Y 398.135,Z 649.494,A -85,B 0,C 180,E1 -11422.902,E2 -11422.902} C_VEL
LIN {X 0,Y 397.627,Z 653.388,A -85,B 0,C 180,E1 -11424.422,E2 -11424.422} C_VEL
LIN {X 0,Y 397.299,Z 656.255,A -85,B 0,C 180,E1 -11425.943,E2 -11425.943} C_VEL
LIN {X 0,Y 397.305,Z 657.607,A -85,B 0,C 180,E1 -11426.958,E2 -11426.958} C_VEL
LIN {X 0,Y 397.137,Z 658.591,A -85,B 0,C 180,E1 -11427.972,E2 -11427.972} C_VEL
LIN {X 0,Y 397.208,Z 659.174,A -85,B 0,C 180,E1 -11428.986,E2 -11428.986} C_VEL
LIN {X 0,Y 397.191,Z 659.403,A -85,B 0,C 180,E1 -11430,E2 -11430} C_VEL
LIN {X 0,Y 397.208,Z 659.218,A -85,B 0,C 180,E1 -11431.014,E2 -11431.014} C_VEL
LIN {X 0,Y 397.136,Z 658.665,A -85,B 0,C 180,E1 -11432.028,E2 -11432.028} C_VEL
LIN {X 0,Y 397.302,Z 657.71,A -85,B 0,C 180,E1 -11433.042,E2 -11433.042} C_VEL
LIN {X 0,Y 397.322,Z 656.025,A -85,B 0,C 180,E1 -11434.274,E2 -11434.274} C_VEL
LIN {X 0,Y 397.676,Z 652.431,A -85,B 0,C 180,E1 -11436.087,E2 -11436.087} C_VEL
LIN {X 0,Y 398.237,Z 648.246,A -85,B 0,C 180,E1 -11437.606,E2 -11437.606} C_VEL
LIN {X 0,Y 398.408,Z 645.55,A -85,B 0,C 180,E1 -11438.425,E2 -11438.425} C_VEL
LIN {X 0,Y 397.989,Z 642.907,A -85,B 0,C 180,E1 -11439.184,E2 -11439.184} C_VEL
LIN {X 0,Y 395.74,Z 638.351,A -85,B 0,C 180,E1 -11440.414,E2 -11440.414} C_VEL
LIN {X 0,Y 393.52,Z 633.183,A -85,B 0,C 180,E1 -11441.598,E2 -11441.598} C_VEL
LIN {X 0,Y 393.143,Z 629.547,A -85,B 0,C 180,E1 -11442.276,E2 -11442.276} C_VEL
LIN {X 0,Y 393.89,Z 620.319,A -85,B 0,C 180,E1 -11443.675,E2 -11443.675} C_VEL
LIN {X 0,Y 394.641,Z 612.011,A -85,B 0,C 180,E1 -11444.7,E2 -11444.7} C_VEL
LIN {X 0,Y 395.422,Z 601.651,A -85,B 0,C 180,E1 -11445.749,E2 -11445.749} C_VEL
LIN {X 0,Y 395.962,Z 591.014,A -85,B 0,C 180,E1 -11446.617,E2 -11446.617} C_VEL
LIN {X 0,Y 396.5,Z 579.577,A -85,B 0,C 180,E1 -11447.337,E2 -11447.337} C_VEL
LIN {X 0,Y 396.804,Z 567.614,A -85,B 0,C 180,E1 -11447.889,E2 -11447.889} C_VEL
LIN {X 0,Y 396.853,Z 555.922,A -85,B 0,C 180,E1 -11448.254,E2 -11448.254} C_VEL
LIN {X 0,Y 397.264,Z 509.847,A -85,B 0,C 180,E1 -11449.113,E2 -11449.113} C_VEL
LIN {X 0,Y 397.379,Z 494.212,A -85,B 0,C 180,E1 -11449.402,E2 -11449.402} C_VEL
LIN {X 0,Y 390.352,Z 477.024,A -85,B 0,C 180,E1 -11450.134,E2 -11450.134} C_VEL
LIN {X 0,Y 390.138,Z 476.105,A -85,B 0,C 180,E1 -11450.289,E2 -11450.289} C_VEL
LIN {X 0,Y 390.09,Z 475.88,A -85,B 0,C 180,E1 -11453.35,E2 -11453.35} C_VEL
LIN {X 0,Y 390.114,Z 475.861,A -85,B 0,C 180,E1 -11456.767,E2 -11456.767} C_VEL
LIN {X 0,Y 390.039,Z 475.9,A -85,B 0,C 180,E1 -11460.299,E2 -11460.299} C_VEL
LIN {X 0,Y 390.067,Z 475.895,A -85,B 0,C 180,E1 -11464.024,E2 -11464.024} C_VEL
LIN {X 0,Y 390.044,Z 475.89,A -85,B 0,C 180,E1 -11467.55,E2 -11467.55} C_VEL
LIN {X 0,Y 390.054,Z 475.896,A -85,B 0,C 180,E1 -11470.821,E2 -11470.821} C_VEL
LIN {X 0,Y 390.053,Z 475.89,A -85,B 0,C 180,E1 -11473.886,E2 -11473.886} C_VEL
LIN {X 0,Y 390.053,Z 475.9,A -85,B 0,C 180,E1 -11476.789,E2 -11476.789} C_VEL
LIN {X 0,Y 390.052,Z 475.869,A -85,B 0,C 180,E1 -11479.56,E2 -11479.56} C_VEL
LIN {X 0,Y 390.039,Z 475.891,A -85,B 0,C 180,E1 -11482.448,E2 -11482.448} C_VEL
LIN {X 0,Y 390.063,Z 475.89,A -85,B 0,C 180,E1 -11485.975,E2 -11485.975} C_VEL
LIN {X 0,Y 390.045,Z 475.865,A -85,B 0,C 180,E1 -11489.867,E2 -11489.867} C_VEL
LIN {X 0,Y 390.107,Z 475.888,A -85,B 0,C 180,E1 -11493.231,E2 -11493.231} C_VEL
LIN {X 0,Y 390.099,Z 475.888,A -85,B 0,C 180,E1 -11496.75,E2 -11496.75} C_VEL
LIN {X 0,Y 390.096,Z 475.89,A -85,B 0,C 180,E1 -11499.982,E2 -11499.982} C_VEL
LIN {X 0,Y 390.13,Z 475.88,A -85,B 0,C 180,E1 -11503.248,E2 -11503.248} C_VEL
LIN {X 0,Y 390.186,Z 475.878,A -85,B 0,C 180,E1 -11506.561,E2 -11506.561} C_VEL
LIN {X 0,Y 390.197,Z 475.865,A -85,B 0,C 180,E1 -11510.671,E2 -11510.671} C_VEL
LIN {X 0,Y 390.309,Z 475.86,A -85,B 0,C 180,E1 -11512.759,E2 -11512.759} C_VEL
LIN {X 0,Y 390.219,Z 475.874,A -85,B 0,C 180,E1 -11514.833,E2 -11514.833} C_VEL
LIN {X 0,Y 390.412,Z 475.843,A -85,B 0,C 180,E1 -11517.937,E2 -11517.937} C_VEL
LIN {X 0,Y 390.543,Z 475.833,A -85,B 0,C 180,E1 -11520,E2 -11520} C_VEL
LIN {X 0,Y 390.308,Z 475.859,A -85,B 0,C 180,E1 -11523.097,E2 -11523.097} C_VEL
LIN {X 0,Y 390.329,Z 475.859,A -85,B 0,C 180,E1 -11526.202,E2 -11526.202} C_VEL
LIN {X 0,Y 390.197,Z 475.877,A -85,B 0,C 180,E1 -11529.329,E2 -11529.329} C_VEL
LIN {X 0,Y 390.186,Z 475.881,A -85,B 0,C 180,E1 -11533.439,E2 -11533.439} C_VEL
LIN {X 0,Y 390.141,Z 475.873,A -85,B 0,C 180,E1 -11537.308,E2 -11537.308} C_VEL
LIN {X 0,Y 390.079,Z 475.883,A -85,B 0,C 180,E1 -11540.47,E2 -11540.47} C_VEL
LIN {X 0,Y 390.082,Z 475.896,A -85,B 0,C 180,E1 -11543.351,E2 -11543.351} C_VEL
LIN {X 0,Y 390.107,Z 475.872,A -85,B 0,C 180,E1 -11546.769,E2 -11546.769} C_VEL
LIN {X 0,Y 390.046,Z 475.898,A -85,B 0,C 180,E1 -11550.299,E2 -11550.299} C_VEL
LIN {X 0,Y 390.063,Z 475.89,A -85,B 0,C 180,E1 -11554.025,E2 -11554.025} C_VEL
LIN {X 0,Y 390.04,Z 475.894,A -85,B 0,C 180,E1 -11557.552,E2 -11557.552} C_VEL
LIN {X 0,Y 390.052,Z 475.897,A -85,B 0,C 180,E1 -11560.822,E2 -11560.822} C_VEL
LIN {X 0,Y 390.055,Z 475.871,A -85,B 0,C 180,E1 -11563.888,E2 -11563.888} C_VEL
LIN {X 0,Y 390.114,Z 475.891,A -85,B 0,C 180,E1 -11566.799,E2 -11566.799} C_VEL
LIN {X 0,Y 390.074,Z 475.879,A -85,B 0,C 180,E1 -11569.564,E2 -11569.564} C_VEL
LIN {X 0,Y 390.045,Z 475.896,A -85,B 0,C 180,E1 -11572.449,E2 -11572.449} C_VEL
LIN {X 0,Y 390.066,Z 475.889,A -85,B 0,C 180,E1 -11576.046,E2 -11576.046} C_VEL
LIN {X 0,Y 390.132,Z 476.192,A -85,B 0,C 180,E1 -11576.363,E2 -11576.363} C_VEL
LIN {X 0,Y 393.998,Z 492.546,A -85,B 0,C 180,E1 -11579.496,E2 -11579.496} C_VEL
LIN {X 0,Y 395.603,Z 500.416,A -85,B 0,C 180,E1 -11580.925,E2 -11580.925} C_VEL
LIN {X 0,Y 394.345,Z 516.52,A -85,B 0,C 180,E1 -11583.542,E2 -11583.542} C_VEL
LIN {X 0,Y 392.591,Z 540.165,A -85,B 0,C 180,E1 -11587.364,E2 -11587.364} C_VEL
LIN {X 0,Y 391.779,Z 553.172,A -85,B 0,C 180,E1 -11589.457,E2 -11589.457} C_VEL
LIN {X 0,Y 395.265,Z 584.357,A -85,B 0,C 180,E1 -11590.256,E2 -11590.256} C_VEL
LIN {X 0,Y 396.366,Z 597.421,A -85,B 0,C 180,E1 -11590.555,E2 -11590.555} C_VEL
LIN {X 0,Y 395.483,Z 663.968,A -85,B 0,C 180,E1 -11591.781,E2 -11591.781} C_VEL
LIN {X 0,Y 394.828,Z 677.252,A -85,B 0,C 180,E1 -11592.219,E2 -11592.219} C_VEL
LIN {X 0,Y 393.946,Z 690.592,A -85,B 0,C 180,E1 -11592.881,E2 -11592.881} C_VEL
LIN {X 0,Y 393.02,Z 701.818,A -85,B 0,C 180,E1 -11593.642,E2 -11593.642} C_VEL
LIN {X 0,Y 391.976,Z 713.525,A -85,B 0,C 180,E1 -11594.665,E2 -11594.665} C_VEL
LIN {X 0,Y 391.109,Z 724.096,A -85,B 0,C 180,E1 -11595.826,E2 -11595.826} C_VEL
LIN {X 0,Y 390.583,Z 732.826,A -85,B 0,C 180,E1 -11597.002,E2 -11597.002} C_VEL
LIN {X 0,Y 389.887,Z 740.855,A -85,B 0,C 180,E1 -11598.3,E2 -11598.3} C_VEL
LIN {X 0,Y 389.394,Z 748.744,A -85,B 0,C 180,E1 -11599.865,E2 -11599.865} C_VEL
LIN {X 0,Y 389.226,Z 754.179,A -85,B 0,C 180,E1 -11601.172,E2 -11601.172} C_VEL
LIN {X 0,Y 389.223,Z 759.478,A -85,B 0,C 180,E1 -11602.739,E2 -11602.739} C_VEL
LIN {X 0,Y 389.256,Z 763.6,A -85,B 0,C 180,E1 -11604.301,E2 -11604.301} C_VEL
LIN {X 0,Y 389.46,Z 766.672,A -85,B 0,C 180,E1 -11605.861,E2 -11605.861} C_VEL
LIN {X 0,Y 389.47,Z 768.123,A -85,B 0,C 180,E1 -11606.897,E2 -11606.897} C_VEL
LIN {X 0,Y 389.795,Z 769.834,A -85,B 0,C 180,E1 -11608.967,E2 -11608.967} C_VEL
LIN {X 0,Y 389.832,Z 770.062,A -85,B 0,C 180,E1 -11610,E2 -11610} C_VEL
LIN {X 0,Y 389.795,Z 769.832,A -85,B 0,C 180,E1 -11611.033,E2 -11611.033} C_VEL
LIN {X 0,Y 389.47,Z 768.12,A -85,B 0,C 180,E1 -11613.103,E2 -11613.103} C_VEL
LIN {X 0,Y 389.475,Z 766.669,A -85,B 0,C 180,E1 -11614.139,E2 -11614.139} C_VEL
LIN {X 0,Y 389.256,Z 763.589,A -85,B 0,C 180,E1 -11615.699,E2 -11615.699} C_VEL
LIN {X 0,Y 389.223,Z 759.46,A -85,B 0,C 180,E1 -11617.261,E2 -11617.261} C_VEL
LIN {X 0,Y 389.26,Z 753.126,A -85,B 0,C 180,E1 -11619.089,E2 -11619.089} C_VEL
LIN {X 0,Y 389.545,Z 746.254,A -85,B 0,C 180,E1 -11620.657,E2 -11620.657} C_VEL
LIN {X 0,Y 390.036,Z 737.765,A -85,B 0,C 180,E1 -11622.223,E2 -11622.223} C_VEL
LIN {X 0,Y 390.761,Z 729.109,A -85,B 0,C 180,E1 -11623.521,E2 -11623.521} C_VEL
LIN {X 0,Y 391.606,Z 718.444,A -85,B 0,C 180,E1 -11624.817,E2 -11624.817} C_VEL
LIN {X 0,Y 392.478,Z 707.932,A -85,B 0,C 180,E1 -11625.847,E2 -11625.847} C_VEL
LIN {X 0,Y 393.462,Z 696.45,A -85,B 0,C 180,E1 -11626.739,E2 -11626.739} C_VEL
LIN {X 0,Y 394.347,Z 684.679,A -85,B 0,C 180,E1 -11627.435,E2 -11627.435} C_VEL
LIN {X 0,Y 395.146,Z 671.148,A -85,B 0,C 180,E1 -11628,E2 -11628} C_VEL
LIN {X 0,Y 395.537,Z 657.725,A -85,B 0,C 180,E1 -11628.35,E2 -11628.35} C_VEL
LIN {X 0,Y 396.273,Z 594.684,A -85,B 0,C 180,E1 -11629.493,E2 -11629.493} C_VEL
LIN {X 0,Y 392.175,Z 557.18,A -85,B 0,C 180,E1 -11630.405,E2 -11630.405} C_VEL
LIN {X 0,Y 391.743,Z 553.097,A -85,B 0,C 180,E1 -11630.545,E2 -11630.545} C_VEL
LIN {X 0,Y 393.181,Z 531.704,A -85,B 0,C 180,E1 -11633.994,E2 -11633.994} C_VEL
LIN {X 0,Y 395.043,Z 507.92,A -85,B 0,C 180,E1 -11637.839,E2 -11637.839} C_VEL
LIN {X 0,Y 395.602,Z 500.302,A -85,B 0,C 180,E1 -11639.08,E2 -11639.08} C_VEL
LIN {X 0,Y 392.682,Z 486.788,A -85,B 0,C 180,E1 -11641.566,E2 -11641.566} C_VEL
LIN {X 0,Y 390.091,Z 476.016,A -85,B 0,C 180,E1 -11643.68,E2 -11643.68} C_VEL
LIN {X 0,Y 390.057,Z 475.886,A -85,B 0,C 180,E1 -11646.482,E2 -11646.482} C_VEL
LIN {X 0,Y 390.071,Z 475.888,A -85,B 0,C 180,E1 -11649.218,E2 -11649.218} C_VEL
LIN {X 0,Y 390.119,Z 475.892,A -85,B 0,C 180,E1 -11652.386,E2 -11652.386} C_VEL
LIN {X 0,Y 390.058,Z 475.874,A -85,B 0,C 180,E1 -11655.356,E2 -11655.356} C_VEL
LIN {X 0,Y 390.026,Z 475.894,A -85,B 0,C 180,E1 -11658.186,E2 -11658.186} C_VEL
LIN {X 0,Y 390.087,Z 475.886,A -85,B 0,C 180,E1 -11660.907,E2 -11660.907} C_VEL
LIN {X 0,Y 390.08,Z 475.892,A -85,B 0,C 180,E1 -11664.792,E2 -11664.792} C_VEL
LIN {X 0,Y 390.024,Z 475.9,A -85,B 0,C 180,E1 -11668.496,E2 -11668.496} C_VEL
LIN {X 0,Y 390.111,Z 475.88,A -85,B 0,C 180,E1 -11672.069,E2 -11672.069} C_VEL
LIN {X 0,Y 390.072,Z 475.891,A -85,B 0,C 180,E1 -11675.519,E2 -11675.519} C_VEL
LIN {X 0,Y 390.048,Z 475.888,A -85,B 0,C 180,E1 -11678.877,E2 -11678.877} C_VEL
LIN {X 0,Y 390.12,Z 475.869,A -85,B 0,C 180,E1 -11682.166,E2 -11682.166} C_VEL
LIN {X 0,Y 390.135,Z 475.885,A -85,B 0,C 180,E1 -11685.392,E2 -11685.392} C_VEL
LIN {X 0,Y 390.14,Z 475.877,A -85,B 0,C 180,E1 -11688.571,E2 -11688.571} C_VEL
LIN {X 0,Y 390.299,Z 475.866,A -85,B 0,C 180,E1 -11692.031,E2 -11692.031} C_VEL
LIN {X 0,Y 390.225,Z 475.864,A -85,B 0,C 180,E1 -11694.834,E2 -11694.834} C_VEL
LIN {X 0,Y 390.412,Z 475.848,A -85,B 0,C 180,E1 -11697.937,E2 -11697.937} C_VEL
LIN {X 0,Y 390.543,Z 475.835,A -85,B 0,C 180,E1 -11700,E2 -11700} C_VEL
LIN {X 0,Y 390.309,Z 475.856,A -85,B 0,C 180,E1 -11703.097,E2 -11703.097} C_VEL
LIN {X 0,Y 390.302,Z 475.862,A -85,B 0,C 180,E1 -11706.6,E2 -11706.6} C_VEL
LIN {X 0,Y 390.197,Z 475.865,A -85,B 0,C 180,E1 -11709.329,E2 -11709.329} C_VEL
LIN {X 0,Y 390.186,Z 475.878,A -85,B 0,C 180,E1 -11713.439,E2 -11713.439} C_VEL
LIN {X 0,Y 390.141,Z 475.883,A -85,B 0,C 180,E1 -11717.308,E2 -11717.308} C_VEL
LIN {X 0,Y 390.08,Z 475.896,A -85,B 0,C 180,E1 -11720.471,E2 -11720.471} C_VEL
LIN {X 0,Y 390.082,Z 475.89,A -85,B 0,C 180,E1 -11723.351,E2 -11723.351} C_VEL
LIN {X 0,Y 390.107,Z 475.888,A -85,B 0,C 180,E1 -11726.769,E2 -11726.769} C_VEL
LIN {X 0,Y 390.037,Z 475.865,A -85,B 0,C 180,E1 -11730.3,E2 -11730.3} C_VEL
LIN {X 0,Y 390.063,Z 475.889,A -85,B 0,C 180,E1 -11734.025,E2 -11734.025} C_VEL
LIN {X 0,Y 390.039,Z 475.891,A -85,B 0,C 180,E1 -11737.552,E2 -11737.552} C_VEL
LIN {X 0,Y 390.052,Z 475.873,A -85,B 0,C 180,E1 -11740.822,E2 -11740.822} C_VEL
LIN {X 0,Y 390.051,Z 475.896,A -85,B 0,C 180,E1 -11743.887,E2 -11743.887} C_VEL
LIN {X 0,Y 390.056,Z 475.882,A -85,B 0,C 180,E1 -11746.791,E2 -11746.791} C_VEL
LIN {X 0,Y 390.055,Z 475.897,A -85,B 0,C 180,E1 -11749.562,E2 -11749.562} C_VEL
LIN {X 0,Y 390.044,Z 475.888,A -85,B 0,C 180,E1 -11752.45,E2 -11752.45} C_VEL
LIN {X 0,Y 390.067,Z 475.847,A -85,B 0,C 180,E1 -11755.976,E2 -11755.976} C_VEL
LIN {X 0,Y 390.046,Z 475.9,A -85,B 0,C 180,E1 -11759.87,E2 -11759.87} C_VEL
LIN {X 0,Y 390.114,Z 475.861,A -85,B 0,C 180,E1 -11763.233,E2 -11763.233} C_VEL
LIN {X 0,Y 390.107,Z 475.878,A -85,B 0,C 180,E1 -11766.751,E2 -11766.751} C_VEL
LIN {X 0,Y 390.148,Z 476.017,A -85,B 0,C 180,E1 -11769.78,E2 -11769.78} C_VEL
LIN {X 0,Y 390.319,Z 476.87,A -85,B 0,C 180,E1 -11769.957,E2 -11769.957} C_VEL
LIN {X 0,Y 397.389,Z 494.278,A -85,B 0,C 180,E1 -11770.701,E2 -11770.701} C_VEL
LIN {X 0,Y 396.821,Z 557.37,A -85,B 0,C 180,E1 -11771.878,E2 -11771.878} C_VEL
LIN {X 0,Y 396.646,Z 570.775,A -85,B 0,C 180,E1 -11772.337,E2 -11772.337} C_VEL
LIN {X 0,Y 396.284,Z 583.478,A -85,B 0,C 180,E1 -11772.986,E2 -11772.986} C_VEL
LIN {X 0,Y 395.794,Z 594.697,A -85,B 0,C 180,E1 -11773.758,E2 -11773.758} C_VEL
LIN {X 0,Y 394.954,Z 606.276,A -85,B 0,C 180,E1 -11774.784,E2 -11774.784} C_VEL
LIN {X 0,Y 394.174,Z 616.609,A -85,B 0,C 180,E1 -11775.941,E2 -11775.941} C_VEL
LIN {X 0,Y 393.47,Z 625.037,A -85,B 0,C 180,E1 -11777.099,E2 -11777.099} C_VEL
LIN {X 0,Y 392.838,Z 632.777,A -85,B 0,C 180,E1 -11778.389,E2 -11778.389} C_VEL
LIN {X 0,Y 392.057,Z 640.46,A -85,B 0,C 180,E1 -11779.961,E2 -11779.961} C_VEL
LIN {X 0,Y 391.504,Z 646.214,A -85,B 0,C 180,E1 -11781.43,E2 -11781.43} C_VEL
LIN {X 0,Y 391.163,Z 650.484,A -85,B 0,C 180,E1 -11782.775,E2 -11782.775} C_VEL
LIN {X 0,Y 390.632,Z 654.378,A -85,B 0,C 180,E1 -11784.321,E2 -11784.321} C_VEL
LIN {X 0,Y 390.287,Z 657.245,A -85,B 0,C 180,E1 -11785.87,E2 -11785.87} C_VEL
LIN {X 0,Y 390.287,Z 658.596,A -85,B 0,C 180,E1 -11786.903,E2 -11786.903} C_VEL
LIN {X 0,Y 390.115,Z 659.58,A -85,B 0,C 180,E1 -11787.935,E2 -11787.935} C_VEL
LIN {X 0,Y 390.184,Z 660.162,A -85,B 0,C 180,E1 -11788.968,E2 -11788.968} C_VEL
LIN {X 0,Y 390.166,Z 660.39,A -85,B 0,C 180,E1 -11790,E2 -11790} C_VEL
LIN {X 0,Y 390.184,Z 660.206,A -85,B 0,C 180,E1 -11791.032,E2 -11791.032} C_VEL
LIN {X 0,Y 390.114,Z 659.652,A -85,B 0,C 180,E1 -11792.065,E2 -11792.065} C_VEL
LIN {X 0,Y 390.284,Z 658.697,A -85,B 0,C 180,E1 -11793.097,E2 -11793.097} C_VEL
LIN {X 0,Y 390.277,Z 657.393,A -85,B 0,C 180,E1 -11794.131,E2 -11794.131} C_VEL
LIN {X 0,Y 390.624,Z 654.58,A -85,B 0,C 180,E1 -11795.679,E2 -11795.679} C_VEL
LIN {X 0,Y 391.14,Z 650.757,A -85,B 0,C 180,E1 -11797.225,E2 -11797.225} C_VEL
LIN {X 0,Y 391.519,Z 645.682,A -85,B 0,C 180,E1 -11798.828,E2 -11798.828} C_VEL
LIN {X 0,Y 392.154,Z 639.656,A -85,B 0,C 180,E1 -11800.324,E2 -11800.324} C_VEL
LIN {X 0,Y 392.955,Z 631.878,A -85,B 0,C 180,E1 -11801.869,E2 -11801.869} C_VEL
LIN {X 0,Y 393.143,Z 629.547,A -85,B 0,C 180,E1 -11802.276,E2 -11802.276} C_VEL
LIN {X 0,Y 392.757,Z 625.743,A -85,B 0,C 180,E1 -11802.933,E2 -11802.933} C_VEL
LIN {X 0,Y 390.549,Z 619.37,A -85,B 0,C 180,E1 -11803.999,E2 -11803.999} C_VEL
LIN {X 0,Y 388.441,Z 612.492,A -85,B 0,C 180,E1 -11804.993,E2 -11804.993} C_VEL
LIN {X 0,Y 388.195,Z 607.853,A -85,B 0,C 180,E1 -11805.526,E2 -11805.526} C_VEL
LIN {X 0,Y 388.998,Z 597.205,A -85,B 0,C 180,E1 -11806.505,E2 -11806.505} C_VEL
LIN {X 0,Y 389.608,Z 586.07,A -85,B 0,C 180,E1 -11807.315,E2 -11807.315} C_VEL
LIN {X 0,Y 389.944,Z 573.286,A -85,B 0,C 180,E1 -11808.011,E2 -11808.011} C_VEL
LIN {X 0,Y 390.116,Z 560.678,A -85,B 0,C 180,E1 -11808.478,E2 -11808.478} C_VEL
LIN {X 0,Y 390.177,Z 536.364,A -85,B 0,C 180,E1 -11808.984,E2 -11808.984} C_VEL
LIN {X 0,Y 390.684,Z 495.795,A -85,B 0,C 180,E1 -11809.736,E2 -11809.736} C_VEL
LIN {X 0,Y 383.262,Z 477.86,A -85,B 0,C 180,E1 -11810.528,E2 -11810.528} C_VEL
LIN {X 0,Y 383.052,Z 476.9,A -85,B 0,C 180,E1 -11810.717,E2 -11810.717} C_VEL
LIN {X 0,Y 383.035,Z 476.767,A -85,B 0,C 180,E1 -11813.807,E2 -11813.807} C_VEL
LIN {X 0,Y 383.057,Z 476.738,A -85,B 0,C 180,E1 -11817.301,E2 -11817.301} C_VEL
LIN {X 0,Y 382.982,Z 476.78,A -85,B 0,C 180,E1 -11820.918,E2 -11820.918} C_VEL
LIN {X 0,Y 383.017,Z 476.776,A -85,B 0,C 180,E1 -11824.667,E2 -11824.667} C_VEL
LIN {X 0,Y 383,Z 476.771,A -85,B 0,C 180,E1 -11827.903,E2 -11827.903} C_VEL
LIN {X 0,Y 382.982,Z 476.768,A -85,B 0,C 180,E1 -11831.346,E2 -11831.346} C_VEL
LIN {X 0,Y 382.994,Z 476.769,A -85,B 0,C 180,E1 -11834.303,E2 -11834.303} C_VEL
LIN {X 0,Y 383.006,Z 476.773,A -85,B 0,C 180,E1 -11837.239,E2 -11837.239} C_VEL
LIN {X 0,Y 383.009,Z 476.744,A -85,B 0,C 180,E1 -11840.413,E2 -11840.413} C_VEL
LIN {X 0,Y 383.021,Z 476.772,A -85,B 0,C 180,E1 -11844.044,E2 -11844.044} C_VEL
LIN {X 0,Y 382.982,Z 476.755,A -85,B 0,C 180,E1 -11847.577,E2 -11847.577} C_VEL
LIN {X 0,Y 382.991,Z 476.747,A -85,B 0,C 180,E1 -11850.3,E2 -11850.3} C_VEL
LIN {X 0,Y 383.05,Z 476.761,A -85,B 0,C 180,E1 -11852.697,E2 -11852.697} C_VEL
LIN {X 0,Y 383.026,Z 476.767,A -85,B 0,C 180,E1 -11856.192,E2 -11856.192} C_VEL
LIN {X 0,Y 383.048,Z 476.771,A -85,B 0,C 180,E1 -11859.598,E2 -11859.598} C_VEL
LIN {X 0,Y 383.097,Z 476.759,A -85,B 0,C 180,E1 -11862.931,E2 -11862.931} C_VEL
LIN {X 0,Y 383.117,Z 476.759,A -85,B 0,C 180,E1 -11866.464,E2 -11866.464} C_VEL
LIN {X 0,Y 383.143,Z 476.743,A -85,B 0,C 180,E1 -11870.498,E2 -11870.498} C_VEL
LIN {X 0,Y 383.264,Z 476.737,A -85,B 0,C 180,E1 -11872.625,E2 -11872.625} C_VEL
LIN {X 0,Y 383.191,Z 476.749,A -85,B 0,C 180,E1 -11874.738,E2 -11874.738} C_VEL
LIN {X 0,Y 383.379,Z 476.718,A -85,B 0,C 180,E1 -11877.899,E2 -11877.899} C_VEL
LIN {X 0,Y 383.512,Z 476.709,A -85,B 0,C 180,E1 -11880,E2 -11880} C_VEL
LIN {X 0,Y 383.245,Z 476.738,A -85,B 0,C 180,E1 -11883.154,E2 -11883.154} C_VEL
LIN {X 0,Y 383.283,Z 476.736,A -85,B 0,C 180,E1 -11886.316,E2 -11886.316} C_VEL
LIN {X 0,Y 383.143,Z 476.753,A -85,B 0,C 180,E1 -11889.502,E2 -11889.502} C_VEL
LIN {X 0,Y 383.117,Z 476.763,A -85,B 0,C 180,E1 -11893.536,E2 -11893.536} C_VEL
LIN {X 0,Y 383.086,Z 476.749,A -85,B 0,C 180,E1 -11897.455,E2 -11897.455} C_VEL
LIN {X 0,Y 383.021,Z 476.762,A -85,B 0,C 180,E1 -11900.647,E2 -11900.647} C_VEL
LIN {X 0,Y 383.026,Z 476.773,A -85,B 0,C 180,E1 -11903.808,E2 -11903.808} C_VEL
LIN {X 0,Y 383.073,Z 476.749,A -85,B 0,C 180,E1 -11906.124,E2 -11906.124} C_VEL
LIN {X 0,Y 383.045,Z 476.765,A -85,B 0,C 180,E1 -11908.492,E2 -11908.492} C_VEL
LIN {X 0,Y 383.007,Z 476.765,A -85,B 0,C 180,E1 -11912.15,E2 -11912.15} C_VEL
LIN {X 0,Y 383.013,Z 476.771,A -85,B 0,C 180,E1 -11914.669,E2 -11914.669} C_VEL
LIN {X 0,Y 382.997,Z 476.769,A -85,B 0,C 180,E1 -11917.905,E2 -11917.905} C_VEL
LIN {X 0,Y 382.98,Z 476.779,A -85,B 0,C 180,E1 -11921.348,E2 -11921.348} C_VEL
LIN {X 0,Y 383.003,Z 476.749,A -85,B 0,C 180,E1 -11924.306,E2 -11924.306} C_VEL
LIN {X 0,Y 383.072,Z 476.77,A -85,B 0,C 180,E1 -11927.25,E2 -11927.25} C_VEL
LIN {X 0,Y 383.019,Z 476.761,A -85,B 0,C 180,E1 -11930.413,E2 -11930.413} C_VEL
LIN {X 0,Y 383.024,Z 476.762,A -85,B 0,C 180,E1 -11934.045,E2 -11934.045} C_VEL
LIN {X 0,Y 383.059,Z 476.929,A -85,B 0,C 180,E1 -11935.955,E2 -11935.955} C_VEL
LIN {X 0,Y 386.689,Z 492.164,A -85,B 0,C 180,E1 -11938.966,E2 -11938.966} C_VEL
LIN {X 0,Y 388.706,Z 501.909,A -85,B 0,C 180,E1 -11940.78,E2 -11940.78} C_VEL
LIN {X 0,Y 387.309,Z 518.962,A -85,B 0,C 180,E1 -11943.605,E2 -11943.605} C_VEL
LIN {X 0,Y 385.598,Z 540.834,A -85,B 0,C 180,E1 -11947.214,E2 -11947.214} C_VEL
LIN {X 0,Y 384.843,Z 552.149,A -85,B 0,C 180,E1 -11949.069,E2 -11949.069} C_VEL
LIN {X 0,Y 388.399,Z 583.35,A -85,B 0,C 180,E1 -11949.892,E2 -11949.892} C_VEL
LIN {X 0,Y 389.613,Z 598.349,A -85,B 0,C 180,E1 -11950.24,E2 -11950.24} C_VEL
LIN {X 0,Y 388.695,Z 662.975,A -85,B 0,C 180,E1 -11951.452,E2 -11951.452} C_VEL
LIN {X 0,Y 388.06,Z 676.26,A -85,B 0,C 180,E1 -11951.898,E2 -11951.898} C_VEL
LIN {X 0,Y 387.243,Z 688.471,A -85,B 0,C 180,E1 -11952.507,E2 -11952.507} C_VEL
LIN {X 0,Y 386.15,Z 700.815,A -85,B 0,C 180,E1 -11953.343,E2 -11953.343} C_VEL
LIN {X 0,Y 385.14,Z 712.532,A -85,B 0,C 180,E1 -11954.386,E2 -11954.386} C_VEL
LIN {X 0,Y 384.149,Z 723.438,A -85,B 0,C 180,E1 -11955.607,E2 -11955.607} C_VEL
LIN {X 0,Y 383.595,Z 731.82,A -85,B 0,C 180,E1 -11956.761,E2 -11956.761} C_VEL
LIN {X 0,Y 382.866,Z 739.849,A -85,B 0,C 180,E1 -11958.083,E2 -11958.083} C_VEL
LIN {X 0,Y 382.346,Z 747.738,A -85,B 0,C 180,E1 -11959.676,E2 -11959.676} C_VEL
LIN {X 0,Y 382.171,Z 753.177,A -85,B 0,C 180,E1 -11961.007,E2 -11961.007} C_VEL
LIN {X 0,Y 382.136,Z 758.474,A -85,B 0,C 180,E1 -11962.603,E2 -11962.603} C_VEL
LIN {X 0,Y 382.195,Z 762.603,A -85,B 0,C 180,E1 -11964.196,E2 -11964.196} C_VEL
LIN {X 0,Y 382.387,Z 765.675,A -85,B 0,C 180,E1 -11965.784,E2 -11965.784} C_VEL
LIN {X 0,Y 382.421,Z 767.131,A -85,B 0,C 180,E1 -11966.84,E2 -11966.84} C_VEL
LIN {X 0,Y 382.765,Z 768.845,A -85,B 0,C 180,E1 -11968.948,E2 -11968.948} C_VEL
LIN {X 0,Y 382.809,Z 769.075,A -85,B 0,C 180,E1 -11970,E2 -11970} C_VEL
LIN {X 0,Y 382.765,Z 768.843,A -85,B 0,C 180,E1 -11971.052,E2 -11971.052} C_VEL
LIN {X 0,Y 382.423,Z 767.128,A -85,B 0,C 180,E1 -11973.16,E2 -11973.16} C_VEL
LIN {X 0,Y 382.399,Z 765.671,A -85,B 0,C 180,E1 -11974.216,E2 -11974.216} C_VEL
LIN {X 0,Y 382.195,Z 762.591,A -85,B 0,C 180,E1 -11975.804,E2 -11975.804} C_VEL
LIN {X 0,Y 382.136,Z 758.454,A -85,B 0,C 180,E1 -11977.397,E2 -11977.397} C_VEL
LIN {X 0,Y 382.205,Z 752.12,A -85,B 0,C 180,E1 -11979.259,E2 -11979.259} C_VEL
LIN {X 0,Y 382.518,Z 745.246,A -85,B 0,C 180,E1 -11980.855,E2 -11980.855} C_VEL
LIN {X 0,Y 383.045,Z 736.756,A -85,B 0,C 180,E1 -11982.45,E2 -11982.45} C_VEL
LIN {X 0,Y 383.787,Z 728.098,A -85,B 0,C 180,E1 -11983.772,E2 -11983.772} C_VEL
LIN {X 0,Y 384.676,Z 717.432,A -85,B 0,C 180,E1 -11985.09,E2 -11985.09} C_VEL
LIN {X 0,Y 385.657,Z 706.931,A -85,B 0,C 180,E1 -11986.135,E2 -11986.135} C_VEL
LIN {X 0,Y 386.615,Z 695.439,A -85,B 0,C 180,E1 -11987.045,E2 -11987.045} C_VEL
LIN {X 0,Y 387.585,Z 683.674,A -85,B 0,C 180,E1 -11987.749,E2 -11987.749} C_VEL
LIN {X 0,Y 388.4,Z 670.14,A -85,B 0,C 180,E1 -11988.324,E2 -11988.324} C_VEL
LIN {X 0,Y 388.786,Z 656.704,A -85,B 0,C 180,E1 -11988.68,E2 -11988.68} C_VEL
LIN {X 0,Y 389.573,Z 595.634,A -85,B 0,C 180,E1 -11989.804,E2 -11989.804} C_VEL
LIN {X 0,Y 385.462,Z 557.769,A -85,B 0,C 180,E1 -11990.745,E2 -11990.745} C_VEL
LIN {X 0,Y 384.831,Z 552.076,A -85,B 0,C 180,E1 -11990.932,E2 -11990.932} C_VEL
LIN {X 0,Y 386.494,Z 529.025,A -85,B 0,C 180,E1 -11994.722,E2 -11994.722} C_VEL
LIN {X 0,Y 388.491,Z 505.269,A -85,B 0,C 180,E1 -11998.645,E2 -11998.645} C_VEL
LIN {X 0,Y 388.739,Z 501.843,A -85,B 0,C 180,E1 -11999.217,E2 -11999.217} C_VEL
LIN {X 0,Y 385.625,Z 487.559,A -85,B 0,C 180,E1 -12001.905,E2 -12001.905} C_VEL
LIN {X 0,Y 383.038,Z 476.899,A -85,B 0,C 180,E1 -12004.047,E2 -12004.047} C_VEL
LIN {X 0,Y 382.996,Z 476.77,A -85,B 0,C 180,E1 -12007.268,E2 -12007.268} C_VEL
LIN {X 0,Y 383.018,Z 476.758,A -85,B 0,C 180,E1 -12009.956,E2 -12009.956} C_VEL
LIN {X 0,Y 383.062,Z 476.771,A -85,B 0,C 180,E1 -12012.788,E2 -12012.788} C_VEL
LIN {X 0,Y 383.003,Z 476.749,A -85,B 0,C 180,E1 -12015.79,E2 -12015.79} C_VEL
LIN {X 0,Y 382.984,Z 476.779,A -85,B 0,C 180,E1 -12018.795,E2 -12018.795} C_VEL
LIN {X 0,Y 382.997,Z 476.769,A -85,B 0,C 180,E1 -12022.095,E2 -12022.095} C_VEL
LIN {X 0,Y 383.012,Z 476.77,A -85,B 0,C 180,E1 -12025.331,E2 -12025.331} C_VEL
LIN {X 0,Y 382.984,Z 476.777,A -85,B 0,C 180,E1 -12029.081,E2 -12029.081} C_VEL
LIN {X 0,Y 383.05,Z 476.752,A -85,B 0,C 180,E1 -12032.698,E2 -12032.698} C_VEL
LIN {X 0,Y 383.045,Z 476.767,A -85,B 0,C 180,E1 -12035.039,E2 -12035.039} C_VEL
LIN {X 0,Y 382.985,Z 476.772,A -85,B 0,C 180,E1 -12038.469,E2 -12038.469} C_VEL
LIN {X 0,Y 383.055,Z 476.746,A -85,B 0,C 180,E1 -12041.826,E2 -12041.826} C_VEL
LIN {X 0,Y 383.101,Z 476.762,A -85,B 0,C 180,E1 -12045.118,E2 -12045.118} C_VEL
LIN {X 0,Y 383.089,Z 476.756,A -85,B 0,C 180,E1 -12048.358,E2 -12048.358} C_VEL
LIN {X 0,Y 383.256,Z 476.743,A -85,B 0,C 180,E1 -12051.975,E2 -12051.975} C_VEL
LIN {X 0,Y 383.197,Z 476.741,A -85,B 0,C 180,E1 -12054.738,E2 -12054.738} C_VEL
LIN {X 0,Y 383.38,Z 476.724,A -85,B 0,C 180,E1 -12057.899,E2 -12057.899} C_VEL
LIN {X 0,Y 383.512,Z 476.711,A -85,B 0,C 180,E1 -12060,E2 -12060} C_VEL
LIN {X 0,Y 383.245,Z 476.736,A -85,B 0,C 180,E1 -12063.154,E2 -12063.154} C_VEL
LIN {X 0,Y 383.262,Z 476.74,A -85,B 0,C 180,E1 -12066.59,E2 -12066.59} C_VEL
LIN {X 0,Y 383.143,Z 476.743,A -85,B 0,C 180,E1 -12069.502,E2 -12069.502} C_VEL
LIN {X 0,Y 383.117,Z 476.758,A -85,B 0,C 180,E1 -12073.536,E2 -12073.536} C_VEL
LIN {X 0,Y 383.087,Z 476.76,A -85,B 0,C 180,E1 -12077.455,E2 -12077.455} C_VEL
LIN {X 0,Y 383.021,Z 476.773,A -85,B 0,C 180,E1 -12080.647,E2 -12080.647} C_VEL
LIN {X 0,Y 383.026,Z 476.767,A -85,B 0,C 180,E1 -12083.808,E2 -12083.808} C_VEL
LIN {X 0,Y 383.05,Z 476.761,A -85,B 0,C 180,E1 -12087.303,E2 -12087.303} C_VEL
LIN {X 0,Y 382.98,Z 476.742,A -85,B 0,C 180,E1 -12090.919,E2 -12090.919} C_VEL
LIN {X 0,Y 383.013,Z 476.772,A -85,B 0,C 180,E1 -12094.669,E2 -12094.669} C_VEL
LIN {X 0,Y 382.995,Z 476.767,A -85,B 0,C 180,E1 -12097.905,E2 -12097.905} C_VEL
LIN {X 0,Y 382.979,Z 476.761,A -85,B 0,C 180,E1 -12101.348,E2 -12101.348} C_VEL
LIN {X 0,Y 382.993,Z 476.777,A -85,B 0,C 180,E1 -12104.304,E2 -12104.304} C_VEL
LIN {X 0,Y 383.007,Z 476.757,A -85,B 0,C 180,E1 -12107.241,E2 -12107.241} C_VEL
LIN {X 0,Y 383.015,Z 476.774,A -85,B 0,C 180,E1 -12110.414,E2 -12110.414} C_VEL
LIN {X 0,Y 383.025,Z 476.734,A -85,B 0,C 180,E1 -12114.045,E2 -12114.045} C_VEL
LIN {X 0,Y 382.986,Z 476.754,A -85,B 0,C 180,E1 -12117.579,E2 -12117.579} C_VEL
LIN {X 0,Y 382.992,Z 476.779,A -85,B 0,C 180,E1 -12120.301,E2 -12120.301} C_VEL
LIN {X 0,Y 383.081,Z 476.744,A -85,B 0,C 180,E1 -12124.022,E2 -12124.022} C_VEL
LIN {X 0,Y 383.009,Z 476.755,A -85,B 0,C 180,E1 -12127.336,E2 -12127.336} C_VEL
LIN {X 0,Y 383.076,Z 476.962,A -85,B 0,C 180,E1 -12129.409,E2 -12129.409} C_VEL
LIN {X 0,Y 383.365,Z 478.108,A -85,B 0,C 180,E1 -12129.593,E2 -12129.593} C_VEL
LIN {X 0,Y 390.694,Z 495.808,A -85,B 0,C 180,E1 -12130.367,E2 -12130.367} C_VEL
LIN {X 0,Y 390.118,Z 558.427,A -85,B 0,C 180,E1 -12131.557,E2 -12131.557} C_VEL
LIN {X 0,Y 389.958,Z 571.779,A -85,B 0,C 180,E1 -12132.024,E2 -12132.024} C_VEL
LIN {X 0,Y 389.607,Z 583.358,A -85,B 0,C 180,E1 -12132.617,E2 -12132.617} C_VEL
LIN {X 0,Y 389.094,Z 594.598,A -85,B 0,C 180,E1 -12133.384,E2 -12133.384} C_VEL
LIN {X 0,Y 388.274,Z 605.999,A -85,B 0,C 180,E1 -12134.381,E2 -12134.381} C_VEL
LIN {X 0,Y 387.414,Z 616.556,A -85,B 0,C 180,E1 -12135.556,E2 -12135.556} C_VEL
LIN {X 0,Y 386.622,Z 626.028,A -85,B 0,C 180,E1 -12136.867,E2 -12136.867} C_VEL
LIN {X 0,Y 385.957,Z 633.768,A -85,B 0,C 180,E1 -12138.179,E2 -12138.179} C_VEL
LIN {X 0,Y 385.139,Z 641.45,A -85,B 0,C 180,E1 -12139.778,E2 -12139.778} C_VEL
LIN {X 0,Y 384.556,Z 647.204,A -85,B 0,C 180,E1 -12141.274,E2 -12141.274} C_VEL
LIN {X 0,Y 384.192,Z 651.473,A -85,B 0,C 180,E1 -12142.643,E2 -12142.643} C_VEL
LIN {X 0,Y 383.638,Z 655.367,A -85,B 0,C 180,E1 -12144.217,E2 -12144.217} C_VEL
LIN {X 0,Y 383.274,Z 658.234,A -85,B 0,C 180,E1 -12145.794,E2 -12145.794} C_VEL
LIN {X 0,Y 383.27,Z 659.585,A -85,B 0,C 180,E1 -12146.847,E2 -12146.847} C_VEL
LIN {X 0,Y 383.092,Z 660.568,A -85,B 0,C 180,E1 -12147.897,E2 -12147.897} C_VEL
LIN {X 0,Y 383.16,Z 661.15,A -85,B 0,C 180,E1 -12148.949,E2 -12148.949} C_VEL
LIN {X 0,Y 383.142,Z 661.378,A -85,B 0,C 180,E1 -12150,E2 -12150} C_VEL
LIN {X 0,Y 383.16,Z 661.194,A -85,B 0,C 180,E1 -12151.051,E2 -12151.051} C_VEL
LIN {X 0,Y 383.092,Z 660.64,A -85,B 0,C 180,E1 -12152.103,E2 -12152.103} C_VEL
LIN {X 0,Y 383.267,Z 659.685,A -85,B 0,C 180,E1 -12153.153,E2 -12153.153} C_VEL
LIN {X 0,Y 383.265,Z 658.38,A -85,B 0,C 180,E1 -12154.206,E2 -12154.206} C_VEL
LIN {X 0,Y 383.63,Z 655.568,A -85,B 0,C 180,E1 -12155.783,E2 -12155.783} C_VEL
LIN {X 0,Y 384.168,Z 651.743,A -85,B 0,C 180,E1 -12157.357,E2 -12157.357} C_VEL
LIN {X 0,Y 384.576,Z 646.668,A -85,B 0,C 180,E1 -12158.989,E2 -12158.989} C_VEL
LIN {X 0,Y 385.242,Z 640.642,A -85,B 0,C 180,E1 -12160.511,E2 -12160.511} C_VEL
LIN {X 0,Y 386.08,Z 632.864,A -85,B 0,C 180,E1 -12162.083,E2 -12162.083} C_VEL
LIN {X 0,Y 386.904,Z 623.195,A -85,B 0,C 180,E1 -12163.659,E2 -12163.659} C_VEL
LIN {X 0,Y 387.713,Z 614.155,A -85,B 0,C 180,E1 -12164.835,E2 -12164.835} C_VEL
LIN {X 0,Y 388.195,Z 607.853,A -85,B 0,C 180,E1 -12165.526,E2 -12165.526} C_VEL
LIN {X 0,Y 387.943,Z 603.053,A -85,B 0,C 180,E1 -12166.034,E2 -12166.034} C_VEL
LIN {X 0,Y 385.805,Z 595.158,A -85,B 0,C 180,E1 -12166.869,E2 -12166.869} C_VEL
LIN {X 0,Y 383.548,Z 586.904,A -85,B 0,C 180,E1 -12167.611,E2 -12167.611} C_VEL
LIN {X 0,Y 383.093,Z 581.523,A -85,B 0,C 180,E1 -12167.965,E2 -12167.965} C_VEL
LIN {X 0,Y 383.42,Z 569.569,A -85,B 0,C 180,E1 -12168.536,E2 -12168.536} C_VEL
LIN {X 0,Y 383.49,Z 557.861,A -85,B 0,C 180,E1 -12168.914,E2 -12168.914} C_VEL
LIN {X 0,Y 383.883,Z 513.744,A -85,B 0,C 180,E1 -12169.768,E2 -12169.768} C_VEL
LIN {X 0,Y 384.071,Z 497.53,A -85,B 0,C 180,E1 -12170.075,E2 -12170.075} C_VEL
LIN {X 0,Y 376.801,Z 480.149,A -85,B 0,C 180,E1 -12170.85,E2 -12170.85} C_VEL
LIN {X 0,Y 376.104,Z 478.248,A -85,B 0,C 180,E1 -12170.993,E2 -12170.993} C_VEL
LIN {X 0,Y 375.981,Z 477.701,A -85,B 0,C 180,E1 -12171.183,E2 -12171.183} C_VEL
LIN {X 0,Y 375.995,Z 477.65,A -85,B 0,C 180,E1 -12174.281,E2 -12174.281} C_VEL
LIN {X 0,Y 376.02,Z 477.615,A -85,B 0,C 180,E1 -12176.651,E2 -12176.651} C_VEL
LIN {X 0,Y 375.964,Z 477.653,A -85,B 0,C 180,E1 -12180.312,E2 -12180.312} C_VEL
LIN {X 0,Y 375.959,Z 477.652,A -85,B 0,C 180,E1 -12184.111,E2 -12184.111} C_VEL
LIN {X 0,Y 375.953,Z 477.642,A -85,B 0,C 180,E1 -12186.74,E2 -12186.74} C_VEL
LIN {X 0,Y 375.987,Z 477.65,A -85,B 0,C 180,E1 -12189.97,E2 -12189.97} C_VEL
LIN {X 0,Y 375.928,Z 477.647,A -85,B 0,C 180,E1 -12193.765,E2 -12193.765} C_VEL
LIN {X 0,Y 375.931,Z 477.66,A -85,B 0,C 180,E1 -12196.81,E2 -12196.81} C_VEL
LIN {X 0,Y 375.957,Z 477.622,A -85,B 0,C 180,E1 -12200.536,E2 -12200.536} C_VEL
LIN {X 0,Y 375.959,Z 477.655,A -85,B 0,C 180,E1 -12203.495,E2 -12203.495} C_VEL
LIN {X 0,Y 375.954,Z 477.647,A -85,B 0,C 180,E1 -12205.888,E2 -12205.888} C_VEL
LIN {X 0,Y 375.962,Z 477.616,A -85,B 0,C 180,E1 -12209.687,E2 -12209.687} C_VEL
LIN {X 0,Y 375.996,Z 477.638,A -85,B 0,C 180,E1 -12212.141,E2 -12212.141} C_VEL
LIN {X 0,Y 375.999,Z 477.646,A -85,B 0,C 180,E1 -12214.538,E2 -12214.538} C_VEL
LIN {X 0,Y 375.956,Z 477.644,A -85,B 0,C 180,E1 -12218.045,E2 -12218.045} C_VEL
LIN {X 0,Y 376.001,Z 477.647,A -85,B 0,C 180,E1 -12221.473,E2 -12221.473} C_VEL
LIN {X 0,Y 376.05,Z 477.631,A -85,B 0,C 180,E1 -12224.832,E2 -12224.832} C_VEL
LIN {X 0,Y 376.042,Z 477.639,A -85,B 0,C 180,E1 -12228.136,E2 -12228.136} C_VEL
LIN {X 0,Y 376.249,Z 477.612,A -85,B 0,C 180,E1 -12231.877,E2 -12231.877} C_VEL
LIN {X 0,Y 376.164,Z 477.624,A -85,B 0,C 180,E1 -12234.64,E2 -12234.64} C_VEL
LIN {X 0,Y 376.345,Z 477.593,A -85,B 0,C 180,E1 -12237.86,E2 -12237.86} C_VEL
LIN {X 0,Y 376.482,Z 477.585,A -85,B 0,C 180,E1 -12240,E2 -12240} C_VEL
LIN {X 0,Y 376.183,Z 477.616,A -85,B 0,C 180,E1 -12243.213,E2 -12243.213} C_VEL
LIN {X 0,Y 376.24,Z 477.614,A -85,B 0,C 180,E1 -12246.435,E2 -12246.435} C_VEL
LIN {X 0,Y 376.111,Z 477.626,A -85,B 0,C 180,E1 -12249.682,E2 -12249.682} C_VEL
LIN {X 0,Y 376.081,Z 477.641,A -85,B 0,C 180,E1 -12253.658,E2 -12253.658} C_VEL
LIN {X 0,Y 376.035,Z 477.624,A -85,B 0,C 180,E1 -12257.607,E2 -12257.607} C_VEL
LIN {X 0,Y 375.971,Z 477.64,A -85,B 0,C 180,E1 -12260.833,E2 -12260.833} C_VEL
LIN {X 0,Y 375.986,Z 477.646,A -85,B 0,C 180,E1 -12264.282,E2 -12264.282} C_VEL
LIN {X 0,Y 376.013,Z 477.626,A -85,B 0,C 180,E1 -12266.653,E2 -12266.653} C_VEL
LIN {X 0,Y 375.975,Z 477.647,A -85,B 0,C 180,E1 -12269.079,E2 -12269.079} C_VEL
LIN {X 0,Y 375.944,Z 477.643,A -85,B 0,C 180,E1 -12272.829,E2 -12272.829} C_VEL
LIN {X 0,Y 375.953,Z 477.654,A -85,B 0,C 180,E1 -12275.416,E2 -12275.416} C_VEL
LIN {X 0,Y 375.971,Z 477.643,A -85,B 0,C 180,E1 -12278.272,E2 -12278.272} C_VEL
LIN {X 0,Y 375.93,Z 477.652,A -85,B 0,C 180,E1 -12281.602,E2 -12281.602} C_VEL
LIN {X 0,Y 375.976,Z 477.634,A -85,B 0,C 180,E1 -12285.261,E2 -12285.261} C_VEL
LIN {X 0,Y 375.987,Z 477.642,A -85,B 0,C 180,E1 -12288.391,E2 -12288.391} C_VEL
LIN {X 0,Y 375.965,Z 477.655,A -85,B 0,C 180,E1 -12291.913,E2 -12291.913} C_VEL
LIN {X 0,Y 375.996,Z 477.812,A -85,B 0,C 180,E1 -12295.576,E2 -12295.576} C_VEL
LIN {X 0,Y 379.396,Z 491.941,A -85,B 0,C 180,E1 -12298.443,E2 -12298.443} C_VEL
LIN {X 0,Y 381.691,Z 502.663,A -85,B 0,C 180,E1 -12300.493,E2 -12300.493} C_VEL
LIN {X 0,Y 381.499,Z 507.816,A -85,B 0,C 180,E1 -12301.382,E2 -12301.382} C_VEL
LIN {X 0,Y 379.36,Z 532.332,A -85,B 0,C 180,E1 -12305.512,E2 -12305.512} C_VEL
LIN {X 0,Y 377.946,Z 551.123,A -85,B 0,C 180,E1 -12308.668,E2 -12308.668} C_VEL
LIN {X 0,Y 381.588,Z 583.02,A -85,B 0,C 180,E1 -12309.53,E2 -12309.53} C_VEL
LIN {X 0,Y 382.925,Z 598.185,A -85,B 0,C 180,E1 -12309.896,E2 -12309.896} C_VEL
LIN {X 0,Y 381.968,Z 661.99,A -85,B 0,C 180,E1 -12311.113,E2 -12311.113} C_VEL
LIN {X 0,Y 381.283,Z 675.265,A -85,B 0,C 180,E1 -12311.565,E2 -12311.565} C_VEL
LIN {X 0,Y 380.467,Z 687.477,A -85,B 0,C 180,E1 -12312.186,E2 -12312.186} C_VEL
LIN {X 0,Y 379.323,Z 699.816,A -85,B 0,C 180,E1 -12313.034,E2 -12313.034} C_VEL
LIN {X 0,Y 378.239,Z 711.527,A -85,B 0,C 180,E1 -12314.094,E2 -12314.094} C_VEL
LIN {X 0,Y 377.222,Z 722.435,A -85,B 0,C 180,E1 -12315.337,E2 -12315.337} C_VEL
LIN {X 0,Y 376.568,Z 730.974,A -85,B 0,C 180,E1 -12316.534,E2 -12316.534} C_VEL
LIN {X 0,Y 375.844,Z 738.841,A -85,B 0,C 180,E1 -12317.856,E2 -12317.856} C_VEL
LIN {X 0,Y 375.295,Z 746.732,A -85,B 0,C 180,E1 -12319.48,E2 -12319.48} C_VEL
LIN {X 0,Y 375.075,Z 754.057,A -85,B 0,C 180,E1 -12321.379,E2 -12321.379} C_VEL
LIN {X 0,Y 375.089,Z 759.605,A -85,B 0,C 180,E1 -12323.245,E2 -12323.245} C_VEL
LIN {X 0,Y 375.161,Z 762.722,A -85,B 0,C 180,E1 -12324.626,E2 -12324.626} C_VEL
LIN {X 0,Y 375.316,Z 764.679,A -85,B 0,C 180,E1 -12325.705,E2 -12325.705} C_VEL
LIN {X 0,Y 375.371,Z 766.138,A -85,B 0,C 180,E1 -12326.78,E2 -12326.78} C_VEL
LIN {X 0,Y 375.734,Z 767.857,A -85,B 0,C 180,E1 -12328.928,E2 -12328.928} C_VEL
LIN {X 0,Y 375.784,Z 768.087,A -85,B 0,C 180,E1 -12330,E2 -12330} C_VEL
LIN {X 0,Y 375.734,Z 767.854,A -85,B 0,C 180,E1 -12331.072,E2 -12331.072} C_VEL
LIN {X 0,Y 375.373,Z 766.134,A -85,B 0,C 180,E1 -12333.22,E2 -12333.22} C_VEL
LIN {X 0,Y 375.327,Z 764.673,A -85,B 0,C 180,E1 -12334.295,E2 -12334.295} C_VEL
LIN {X 0,Y 375.138,Z 761.592,A -85,B 0,C 180,E1 -12335.914,E2 -12335.914} C_VEL
LIN {X 0,Y 375.062,Z 757.45,A -85,B 0,C 180,E1 -12337.537,E2 -12337.537} C_VEL
LIN {X 0,Y 375.168,Z 751.116,A -85,B 0,C 180,E1 -12339.434,E2 -12339.434} C_VEL
LIN {X 0,Y 375.475,Z 744.236,A -85,B 0,C 180,E1 -12341.061,E2 -12341.061} C_VEL
LIN {X 0,Y 376.078,Z 735.751,A -85,B 0,C 180,E1 -12342.684,E2 -12342.684} C_VEL
LIN {X 0,Y 376.79,Z 726.678,A -85,B 0,C 180,E1 -12344.088,E2 -12344.088} C_VEL
LIN {X 0,Y 377.781,Z 716.424,A -85,B 0,C 180,E1 -12345.372,E2 -12345.372} C_VEL
LIN {X 0,Y 378.801,Z 705.922,A -85,B 0,C 180,E1 -12346.435,E2 -12346.435} C_VEL
LIN {X 0,Y 379.823,Z 694.434,A -85,B 0,C 180,E1 -12347.359,E2 -12347.359} C_VEL
LIN {X 0,Y 380.782,Z 682.661,A -85,B 0,C 180,E1 -12348.077,E2 -12348.077} C_VEL
LIN {X 0,Y 381.658,Z 669.13,A -85,B 0,C 180,E1 -12348.659,E2 -12348.659} C_VEL
LIN {X 0,Y 382.057,Z 655.685,A -85,B 0,C 180,E1 -12349.022,E2 -12349.022} C_VEL
LIN {X 0,Y 382.824,Z 596.119,A -85,B 0,C 180,E1 -12350.139,E2 -12350.139} C_VEL
LIN {X 0,Y 378.923,Z 559.542,A -85,B 0,C 180,E1 -12351.065,E2 -12351.065} C_VEL
LIN {X 0,Y 377.91,Z 551.145,A -85,B 0,C 180,E1 -12351.322,E2 -12351.322} C_VEL
LIN {X 0,Y 379.579,Z 529.483,A -85,B 0,C 180,E1 -12354.953,E2 -12354.953} C_VEL
LIN {X 0,Y 381.484,Z 507.735,A -85,B 0,C 180,E1 -12358.619,E2 -12358.619} C_VEL
LIN {X 0,Y 381.769,Z 502.591,A -85,B 0,C 180,E1 -12359.5,E2 -12359.5} C_VEL
LIN {X 0,Y 378.523,Z 488.159,A -85,B 0,C 180,E1 -12362.289,E2 -12362.289} C_VEL
LIN {X 0,Y 376.009,Z 477.762,A -85,B 0,C 180,E1 -12364.443,E2 -12364.443} C_VEL
LIN {X 0,Y 375.975,Z 477.654,A -85,B 0,C 180,E1 -12368.27,E2 -12368.27} C_VEL
LIN {X 0,Y 375.987,Z 477.643,A -85,B 0,C 180,E1 -12371.609,E2 -12371.609} C_VEL
LIN {X 0,Y 375.965,Z 477.628,A -85,B 0,C 180,E1 -12375.261,E2 -12375.261} C_VEL
LIN {X 0,Y 375.936,Z 477.655,A -85,B 0,C 180,E1 -12379.132,E2 -12379.132} C_VEL
LIN {X 0,Y 375.961,Z 477.644,A -85,B 0,C 180,E1 -12381.911,E2 -12381.911} C_VEL
LIN {X 0,Y 375.974,Z 477.647,A -85,B 0,C 180,E1 -12385.332,E2 -12385.332} C_VEL
LIN {X 0,Y 375.956,Z 477.651,A -85,B 0,C 180,E1 -12388.438,E2 -12388.438} C_VEL
LIN {X 0,Y 375.996,Z 477.636,A -85,B 0,C 180,E1 -12392.141,E2 -12392.141} C_VEL
LIN {X 0,Y 375.999,Z 477.638,A -85,B 0,C 180,E1 -12394.538,E2 -12394.538} C_VEL
LIN {X 0,Y 375.955,Z 477.654,A -85,B 0,C 180,E1 -12398.045,E2 -12398.045} C_VEL
LIN {X 0,Y 376.001,Z 477.623,A -85,B 0,C 180,E1 -12401.473,E2 -12401.473} C_VEL
LIN {X 0,Y 376.05,Z 477.643,A -85,B 0,C 180,E1 -12404.832,E2 -12404.832} C_VEL
LIN {X 0,Y 376.042,Z 477.635,A -85,B 0,C 180,E1 -12408.136,E2 -12408.136} C_VEL
LIN {X 0,Y 376.212,Z 477.62,A -85,B 0,C 180,E1 -12411.918,E2 -12411.918} C_VEL
LIN {X 0,Y 376.169,Z 477.617,A -85,B 0,C 180,E1 -12414.64,E2 -12414.64} C_VEL
LIN {X 0,Y 376.346,Z 477.6,A -85,B 0,C 180,E1 -12417.86,E2 -12417.86} C_VEL
LIN {X 0,Y 376.482,Z 477.587,A -85,B 0,C 180,E1 -12420,E2 -12420} C_VEL
LIN {X 0,Y 376.183,Z 477.615,A -85,B 0,C 180,E1 -12423.213,E2 -12423.213} C_VEL
LIN {X 0,Y 376.227,Z 477.619,A -85,B 0,C 180,E1 -12426.577,E2 -12426.577} C_VEL
LIN {X 0,Y 376.111,Z 477.618,A -85,B 0,C 180,E1 -12429.682,E2 -12429.682} C_VEL
LIN {X 0,Y 376.081,Z 477.635,A -85,B 0,C 180,E1 -12433.658,E2 -12433.658} C_VEL
LIN {X 0,Y 376.035,Z 477.638,A -85,B 0,C 180,E1 -12437.607,E2 -12437.607} C_VEL
LIN {X 0,Y 375.971,Z 477.648,A -85,B 0,C 180,E1 -12440.833,E2 -12440.833} C_VEL
LIN {X 0,Y 375.987,Z 477.646,A -85,B 0,C 180,E1 -12444.282,E2 -12444.282} C_VEL
LIN {X 0,Y 376.013,Z 477.645,A -85,B 0,C 180,E1 -12446.653,E2 -12446.653} C_VEL
LIN {X 0,Y 375.97,Z 477.625,A -85,B 0,C 180,E1 -12449.079,E2 -12449.079} C_VEL
LIN {X 0,Y 375.944,Z 477.635,A -85,B 0,C 180,E1 -12452.829,E2 -12452.829} C_VEL
LIN {X 0,Y 375.953,Z 477.654,A -85,B 0,C 180,E1 -12455.416,E2 -12455.416} C_VEL
LIN {X 0,Y 375.969,Z 477.641,A -85,B 0,C 180,E1 -12458.271,E2 -12458.271} C_VEL
LIN {X 0,Y 375.93,Z 477.643,A -85,B 0,C 180,E1 -12461.602,E2 -12461.602} C_VEL
LIN {X 0,Y 375.925,Z 477.652,A -85,B 0,C 180,E1 -12465.269,E2 -12465.269} C_VEL
LIN {X 0,Y 375.933,Z 477.642,A -85,B 0,C 180,E1 -12468.4,E2 -12468.4} C_VEL
LIN {X 0,Y 375.974,Z 477.646,A -85,B 0,C 180,E1 -12471.73,E2 -12471.73} C_VEL
LIN {X 0,Y 375.979,Z 477.596,A -85,B 0,C 180,E1 -12475.333,E2 -12475.333} C_VEL
LIN {X 0,Y 375.957,Z 477.649,A -85,B 0,C 180,E1 -12478.439,E2 -12478.439} C_VEL
LIN {X 0,Y 375.983,Z 477.623,A -85,B 0,C 180,E1 -12482.141,E2 -12482.141} C_VEL
LIN {X 0,Y 376.007,Z 477.634,A -85,B 0,C 180,E1 -12484.54,E2 -12484.54} C_VEL
LIN {X 0,Y 375.966,Z 477.631,A -85,B 0,C 180,E1 -12488.046,E2 -12488.046} C_VEL
LIN {X 0,Y 376.019,Z 477.852,A -85,B 0,C 180,E1 -12489.006,E2 -12489.006} C_VEL
LIN {X 0,Y 376.194,Z 478.698,A -85,B 0,C 180,E1 -12489.167,E2 -12489.167} C_VEL
LIN {X 0,Y 383.963,Z 497.284,A -85,B 0,C 180,E1 -12490.017,E2 -12490.017} C_VEL
LIN {X 0,Y 383.431,Z 559.814,A -85,B 0,C 180,E1 -12491.234,E2 -12491.234} C_VEL
LIN {X 0,Y 383.268,Z 572.83,A -85,B 0,C 180,E1 -12491.701,E2 -12491.701} C_VEL
LIN {X 0,Y 382.902,Z 584.354,A -85,B 0,C 180,E1 -12492.303,E2 -12492.303} C_VEL
LIN {X 0,Y 382.318,Z 596.687,A -85,B 0,C 180,E1 -12493.169,E2 -12493.169} C_VEL
LIN {X 0,Y 381.405,Z 608.262,A -85,B 0,C 180,E1 -12494.229,E2 -12494.229} C_VEL
LIN {X 0,Y 380.552,Z 618.593,A -85,B 0,C 180,E1 -12495.427,E2 -12495.427} C_VEL
LIN {X 0,Y 379.78,Z 627.02,A -85,B 0,C 180,E1 -12496.626,E2 -12496.626} C_VEL
LIN {X 0,Y 379.08,Z 634.759,A -85,B 0,C 180,E1 -12497.962,E2 -12497.962} C_VEL
LIN {X 0,Y 378.224,Z 642.44,A -85,B 0,C 180,E1 -12499.589,E2 -12499.589} C_VEL
LIN {X 0,Y 377.611,Z 648.193,A -85,B 0,C 180,E1 -12501.112,E2 -12501.112} C_VEL
LIN {X 0,Y 377.223,Z 652.463,A -85,B 0,C 180,E1 -12502.507,E2 -12502.507} C_VEL
LIN {X 0,Y 376.645,Z 656.356,A -85,B 0,C 180,E1 -12504.11,E2 -12504.11} C_VEL
LIN {X 0,Y 376.263,Z 659.223,A -85,B 0,C 180,E1 -12505.715,E2 -12505.715} C_VEL
LIN {X 0,Y 376.252,Z 660.573,A -85,B 0,C 180,E1 -12506.788,E2 -12506.788} C_VEL
LIN {X 0,Y 376.07,Z 661.556,A -85,B 0,C 180,E1 -12507.858,E2 -12507.858} C_VEL
LIN {X 0,Y 376.135,Z 662.138,A -85,B 0,C 180,E1 -12508.929,E2 -12508.929} C_VEL
LIN {X 0,Y 376.116,Z 662.366,A -85,B 0,C 180,E1 -12510,E2 -12510} C_VEL
LIN {X 0,Y 376.135,Z 662.181,A -85,B 0,C 180,E1 -12511.071,E2 -12511.071} C_VEL
LIN {X 0,Y 376.07,Z 661.628,A -85,B 0,C 180,E1 -12512.142,E2 -12512.142} C_VEL
LIN {X 0,Y 376.249,Z 660.673,A -85,B 0,C 180,E1 -12513.212,E2 -12513.212} C_VEL
LIN {X 0,Y 376.253,Z 659.368,A -85,B 0,C 180,E1 -12514.285,E2 -12514.285} C_VEL
LIN {X 0,Y 376.638,Z 656.555,A -85,B 0,C 180,E1 -12515.89,E2 -12515.89} C_VEL
LIN {X 0,Y 377.199,Z 652.73,A -85,B 0,C 180,E1 -12517.494,E2 -12517.494} C_VEL
LIN {X 0,Y 377.636,Z 647.655,A -85,B 0,C 180,E1 -12519.155,E2 -12519.155} C_VEL
LIN {X 0,Y 378.334,Z 641.628,A -85,B 0,C 180,E1 -12520.705,E2 -12520.705} C_VEL
LIN {X 0,Y 379.21,Z 633.849,A -85,B 0,C 180,E1 -12522.306,E2 -12522.306} C_VEL
LIN {X 0,Y 380.077,Z 624.18,A -85,B 0,C 180,E1 -12523.909,E2 -12523.909} C_VEL
LIN {X 0,Y 380.924,Z 615.139,A -85,B 0,C 180,E1 -12525.106,E2 -12525.106} C_VEL
LIN {X 0,Y 381.793,Z 604.643,A -85,B 0,C 180,E1 -12526.227,E2 -12526.227} C_VEL
LIN {X 0,Y 382.513,Z 592.978,A -85,B 0,C 180,E1 -12527.219,E2 -12527.219} C_VEL
LIN {X 0,Y 383.093,Z 581.523,A -85,B 0,C 180,E1 -12527.965,E2 -12527.965} C_VEL
LIN {X 0,Y 382.649,Z 576.023,A -85,B 0,C 180,E1 -12528.289,E2 -12528.289} C_VEL
LIN {X 0,Y 380.145,Z 567.096,A -85,B 0,C 180,E1 -12528.816,E2 -12528.816} C_VEL
LIN {X 0,Y 377.482,Z 558.007,A -85,B 0,C 180,E1 -12529.246,E2 -12529.246} C_VEL
LIN {X 0,Y 376.782,Z 552.259,A -85,B 0,C 180,E1 -12529.408,E2 -12529.408} C_VEL
LIN {X 0,Y 377.445,Z 499.276,A -85,B 0,C 180,E1 -12530.428,E2 -12530.428} C_VEL
LIN {X 0,Y 370,Z 481.517,A -85,B 0,C 180,E1 -12531.244,E2 -12531.244} C_VEL
LIN {X 0,Y 369.065,Z 479.251,A -85,B 0,C 180,E1 -12531.398,E2 -12531.398} C_VEL
LIN {X 0,Y 368.925,Z 478.583,A -85,B 0,C 180,E1 -12531.607,E2 -12531.607} C_VEL
LIN {X 0,Y 368.959,Z 478.527,A -85,B 0,C 180,E1 -12534.775,E2 -12534.775} C_VEL
LIN {X 0,Y 368.963,Z 478.491,A -85,B 0,C 180,E1 -12537.203,E2 -12537.203} C_VEL
LIN {X 0,Y 368.929,Z 478.53,A -85,B 0,C 180,E1 -12540.953,E2 -12540.953} C_VEL
LIN {X 0,Y 368.928,Z 478.53,A -85,B 0,C 180,E1 -12545.001,E2 -12545.001} C_VEL
LIN {X 0,Y 368.908,Z 478.528,A -85,B 0,C 180,E1 -12548.64,E2 -12548.64} C_VEL
LIN {X 0,Y 368.879,Z 478.52,A -85,B 0,C 180,E1 -12552.009,E2 -12552.009} C_VEL
LIN {X 0,Y 368.923,Z 478.53,A -85,B 0,C 180,E1 -12555.182,E2 -12555.182} C_VEL
LIN {X 0,Y 368.879,Z 478.527,A -85,B 0,C 180,E1 -12558.177,E2 -12558.177} C_VEL
LIN {X 0,Y 368.903,Z 478.51,A -85,B 0,C 180,E1 -12561.359,E2 -12561.359} C_VEL
LIN {X 0,Y 368.931,Z 478.529,A -85,B 0,C 180,E1 -12565.146,E2 -12565.146} C_VEL
LIN {X 0,Y 368.924,Z 478.491,A -85,B 0,C 180,E1 -12569.046,E2 -12569.046} C_VEL
LIN {X 0,Y 368.98,Z 478.503,A -85,B 0,C 180,E1 -12571.564,E2 -12571.564} C_VEL
LIN {X 0,Y 368.951,Z 478.528,A -85,B 0,C 180,E1 -12575.224,E2 -12575.224} C_VEL
LIN {X 0,Y 368.913,Z 478.524,A -85,B 0,C 180,E1 -12578.98,E2 -12578.98} C_VEL
LIN {X 0,Y 368.983,Z 478.516,A -85,B 0,C 180,E1 -12582.257,E2 -12582.257} C_VEL
LIN {X 0,Y 369.029,Z 478.514,A -85,B 0,C 180,E1 -12586.227,E2 -12586.227} C_VEL
LIN {X 0,Y 369.06,Z 478.497,A -85,B 0,C 180,E1 -12590.131,E2 -12590.131} C_VEL
LIN {X 0,Y 369.179,Z 478.491,A -85,B 0,C 180,E1 -12592.342,E2 -12592.342} C_VEL
LIN {X 0,Y 369.137,Z 478.499,A -85,B 0,C 180,E1 -12594.537,E2 -12594.537} C_VEL
LIN {X 0,Y 369.31,Z 478.468,A -85,B 0,C 180,E1 -12597.819,E2 -12597.819} C_VEL
LIN {X 0,Y 369.451,Z 478.46,A -85,B 0,C 180,E1 -12600,E2 -12600} C_VEL
LIN {X 0,Y 369.311,Z 478.474,A -85,B 0,C 180,E1 -12602.181,E2 -12602.181} C_VEL
LIN {X 0,Y 369.199,Z 478.491,A -85,B 0,C 180,E1 -12606.558,E2 -12606.558} C_VEL
LIN {X 0,Y 369.059,Z 478.502,A -85,B 0,C 180,E1 -12609.868,E2 -12609.868} C_VEL
LIN {X 0,Y 369.029,Z 478.519,A -85,B 0,C 180,E1 -12613.772,E2 -12613.772} C_VEL
LIN {X 0,Y 368.994,Z 478.498,A -85,B 0,C 180,E1 -12617.769,E2 -12617.769} C_VEL
LIN {X 0,Y 368.903,Z 478.523,A -85,B 0,C 180,E1 -12621.221,E2 -12621.221} C_VEL
LIN {X 0,Y 368.95,Z 478.522,A -85,B 0,C 180,E1 -12624.776,E2 -12624.776} C_VEL
LIN {X 0,Y 368.982,Z 478.517,A -85,B 0,C 180,E1 -12628.436,E2 -12628.436} C_VEL
LIN {X 0,Y 368.895,Z 478.522,A -85,B 0,C 180,E1 -12632.238,E2 -12632.238} C_VEL
LIN {X 0,Y 368.924,Z 478.526,A -85,B 0,C 180,E1 -12635.002,E2 -12635.002} C_VEL
LIN {X 0,Y 368.905,Z 478.525,A -85,B 0,C 180,E1 -12638.641,E2 -12638.641} C_VEL
LIN {X 0,Y 368.877,Z 478.525,A -85,B 0,C 180,E1 -12642.01,E2 -12642.01} C_VEL
LIN {X 0,Y 368.951,Z 478.507,A -85,B 0,C 180,E1 -12645.188,E2 -12645.188} C_VEL
LIN {X 0,Y 368.938,Z 478.521,A -85,B 0,C 180,E1 -12648.187,E2 -12648.187} C_VEL
LIN {X 0,Y 368.911,Z 478.531,A -85,B 0,C 180,E1 -12651.36,E2 -12651.36} C_VEL
LIN {X 0,Y 368.956,Z 478.667,A -85,B 0,C 180,E1 -12655.17,E2 -12655.17} C_VEL
LIN {X 0,Y 371.93,Z 490.939,A -85,B 0,C 180,E1 -12657.737,E2 -12657.737} C_VEL
LIN {X 0,Y 374.724,Z 503.685,A -85,B 0,C 180,E1 -12660.246,E2 -12660.246} C_VEL
LIN {X 0,Y 374.805,Z 506.876,A -85,B 0,C 180,E1 -12660.823,E2 -12660.823} C_VEL
LIN {X 0,Y 372.812,Z 528.168,A -85,B 0,C 180,E1 -12664.488,E2 -12664.488} C_VEL
LIN {X 0,Y 371.073,Z 550.233,A -85,B 0,C 180,E1 -12668.265,E2 -12668.265} C_VEL
LIN {X 0,Y 375.094,Z 585.423,A -85,B 0,C 180,E1 -12669.226,E2 -12669.226} C_VEL
LIN {X 0,Y 376.204,Z 599.691,A -85,B 0,C 180,E1 -12669.57,E2 -12669.57} C_VEL
LIN {X 0,Y 375.248,Z 661.003,A -85,B 0,C 180,E1 -12670.761,E2 -12670.761} C_VEL
LIN {X 0,Y 374.557,Z 674.276,A -85,B 0,C 180,E1 -12671.222,E2 -12671.222} C_VEL
LIN {X 0,Y 373.684,Z 686.481,A -85,B 0,C 180,E1 -12671.851,E2 -12671.851} C_VEL
LIN {X 0,Y 372.493,Z 698.816,A -85,B 0,C 180,E1 -12672.713,E2 -12672.713} C_VEL
LIN {X 0,Y 371.422,Z 710.533,A -85,B 0,C 180,E1 -12673.794,E2 -12673.794} C_VEL
LIN {X 0,Y 370.375,Z 721.111,A -85,B 0,C 180,E1 -12675.017,E2 -12675.017} C_VEL
LIN {X 0,Y 369.528,Z 730.463,A -85,B 0,C 180,E1 -12676.352,E2 -12676.352} C_VEL
LIN {X 0,Y 368.751,Z 739.253,A -85,B 0,C 180,E1 -12677.899,E2 -12677.899} C_VEL
LIN {X 0,Y 368.197,Z 746.88,A -85,B 0,C 180,E1 -12679.553,E2 -12679.553} C_VEL
LIN {X 0,Y 368.007,Z 753.053,A -85,B 0,C 180,E1 -12681.212,E2 -12681.212} C_VEL
LIN {X 0,Y 368.003,Z 757.961,A -85,B 0,C 180,E1 -12682.87,E2 -12682.87} C_VEL
LIN {X 0,Y 368.092,Z 761.724,A -85,B 0,C 180,E1 -12684.522,E2 -12684.522} C_VEL
LIN {X 0,Y 368.248,Z 763.683,A -85,B 0,C 180,E1 -12685.622,E2 -12685.622} C_VEL
LIN {X 0,Y 368.321,Z 765.146,A -85,B 0,C 180,E1 -12686.718,E2 -12686.718} C_VEL
LIN {X 0,Y 368.702,Z 766.868,A -85,B 0,C 180,E1 -12688.908,E2 -12688.908} C_VEL
LIN {X 0,Y 368.76,Z 767.099,A -85,B 0,C 180,E1 -12690,E2 -12690} C_VEL
LIN {X 0,Y 368.702,Z 766.865,A -85,B 0,C 180,E1 -12691.092,E2 -12691.092} C_VEL
LIN {X 0,Y 368.323,Z 765.141,A -85,B 0,C 180,E1 -12693.282,E2 -12693.282} C_VEL
LIN {X 0,Y 368.257,Z 763.675,A -85,B 0,C 180,E1 -12694.378,E2 -12694.378} C_VEL
LIN {X 0,Y 368.078,Z 760.594,A -85,B 0,C 180,E1 -12696.028,E2 -12696.028} C_VEL
LIN {X 0,Y 367.99,Z 756.446,A -85,B 0,C 180,E1 -12697.683,E2 -12697.683} C_VEL
LIN {X 0,Y 368.105,Z 750.108,A -85,B 0,C 180,E1 -12699.617,E2 -12699.617} C_VEL
LIN {X 0,Y 368.457,Z 743.229,A -85,B 0,C 180,E1 -12701.274,E2 -12701.274} C_VEL
LIN {X 0,Y 369.127,Z 734.746,A -85,B 0,C 180,E1 -12702.927,E2 -12702.927} C_VEL
LIN {X 0,Y 369.815,Z 726.068,A -85,B 0,C 180,E1 -12704.303,E2 -12704.303} C_VEL
LIN {X 0,Y 370.825,Z 715.406,A -85,B 0,C 180,E1 -12705.668,E2 -12705.668} C_VEL
LIN {X 0,Y 372.08,Z 703.467,A -85,B 0,C 180,E1 -12706.882,E2 -12706.882} C_VEL
LIN {X 0,Y 373.21,Z 691.479,A -85,B 0,C 180,E1 -12707.818,E2 -12707.818} C_VEL
LIN {X 0,Y 374.228,Z 679.042,A -85,B 0,C 180,E1 -12708.547,E2 -12708.547} C_VEL
LIN {X 0,Y 374.997,Z 666.275,A -85,B 0,C 180,E1 -12709.074,E2 -12709.074} C_VEL
LIN {X 0,Y 375.37,Z 652.869,A -85,B 0,C 180,E1 -12709.41,E2 -12709.41} C_VEL
LIN {X 0,Y 376.078,Z 596.295,A -85,B 0,C 180,E1 -12710.493,E2 -12710.493} C_VEL
LIN {X 0,Y 372.234,Z 560.202,A -85,B 0,C 180,E1 -12711.428,E2 -12711.428} C_VEL
LIN {X 0,Y 371.045,Z 550.184,A -85,B 0,C 180,E1 -12711.729,E2 -12711.729} C_VEL
LIN {X 0,Y 372.783,Z 528.066,A -85,B 0,C 180,E1 -12715.516,E2 -12715.516} C_VEL
LIN {X 0,Y 374.822,Z 506.792,A -85,B 0,C 180,E1 -12719.176,E2 -12719.176} C_VEL
LIN {X 0,Y 374.754,Z 503.577,A -85,B 0,C 180,E1 -12719.754,E2 -12719.754} C_VEL
LIN {X 0,Y 371.086,Z 487.286,A -85,B 0,C 180,E1 -12722.989,E2 -12722.989} C_VEL
LIN {X 0,Y 368.954,Z 478.628,A -85,B 0,C 180,E1 -12724.851,E2 -12724.851} C_VEL
LIN {X 0,Y 368.911,Z 478.53,A -85,B 0,C 180,E1 -12728.64,E2 -12728.64} C_VEL
LIN {X 0,Y 368.939,Z 478.524,A -85,B 0,C 180,E1 -12732.019,E2 -12732.019} C_VEL
LIN {X 0,Y 368.92,Z 478.505,A -85,B 0,C 180,E1 -12735.182,E2 -12735.182} C_VEL
LIN {X 0,Y 368.879,Z 478.527,A -85,B 0,C 180,E1 -12738.177,E2 -12738.177} C_VEL
LIN {X 0,Y 368.905,Z 478.523,A -85,B 0,C 180,E1 -12741.359,E2 -12741.359} C_VEL
LIN {X 0,Y 368.931,Z 478.524,A -85,B 0,C 180,E1 -12745.146,E2 -12745.146} C_VEL
LIN {X 0,Y 368.923,Z 478.529,A -85,B 0,C 180,E1 -12749.046,E2 -12749.046} C_VEL
LIN {X 0,Y 368.982,Z 478.516,A -85,B 0,C 180,E1 -12751.564,E2 -12751.564} C_VEL
LIN {X 0,Y 368.95,Z 478.522,A -85,B 0,C 180,E1 -12755.224,E2 -12755.224} C_VEL
LIN {X 0,Y 368.912,Z 478.519,A -85,B 0,C 180,E1 -12758.98,E2 -12758.98} C_VEL
LIN {X 0,Y 368.983,Z 478.501,A -85,B 0,C 180,E1 -12762.257,E2 -12762.257} C_VEL
LIN {X 0,Y 369.029,Z 478.518,A -85,B 0,C 180,E1 -12766.228,E2 -12766.228} C_VEL
LIN {X 0,Y 369.059,Z 478.503,A -85,B 0,C 180,E1 -12770.132,E2 -12770.132} C_VEL
LIN {X 0,Y 369.199,Z 478.491,A -85,B 0,C 180,E1 -12773.442,E2 -12773.442} C_VEL
LIN {X 0,Y 369.311,Z 478.476,A -85,B 0,C 180,E1 -12777.819,E2 -12777.819} C_VEL
LIN {X 0,Y 369.452,Z 478.463,A -85,B 0,C 180,E1 -12780,E2 -12780} C_VEL
LIN {X 0,Y 369.311,Z 478.47,A -85,B 0,C 180,E1 -12782.181,E2 -12782.181} C_VEL
LIN {X 0,Y 369.199,Z 478.497,A -85,B 0,C 180,E1 -12786.56,E2 -12786.56} C_VEL
LIN {X 0,Y 369.06,Z 478.497,A -85,B 0,C 180,E1 -12789.869,E2 -12789.869} C_VEL
LIN {X 0,Y 369.029,Z 478.513,A -85,B 0,C 180,E1 -12793.773,E2 -12793.773} C_VEL
LIN {X 0,Y 368.994,Z 478.515,A -85,B 0,C 180,E1 -12797.769,E2 -12797.769} C_VEL
LIN {X 0,Y 368.904,Z 478.524,A -85,B 0,C 180,E1 -12801.221,E2 -12801.221} C_VEL
LIN {X 0,Y 368.951,Z 478.528,A -85,B 0,C 180,E1 -12804.776,E2 -12804.776} C_VEL
LIN {X 0,Y 368.98,Z 478.504,A -85,B 0,C 180,E1 -12808.436,E2 -12808.436} C_VEL
LIN {X 0,Y 368.893,Z 478.507,A -85,B 0,C 180,E1 -12812.239,E2 -12812.239} C_VEL
LIN {X 0,Y 368.924,Z 478.531,A -85,B 0,C 180,E1 -12815.002,E2 -12815.002} C_VEL
LIN {X 0,Y 368.903,Z 478.512,A -85,B 0,C 180,E1 -12818.641,E2 -12818.641} C_VEL
